       "LT".TCH_LFT_DN_REL :=         "PDI".EMO AND "PDI".EMS 
                            AND NOT "FLT".TCH_LFT_ERR 
                          //  AND     TCH_LFT_FU_RDY
                            AND NOT "PDI".LS_TCH_DN
                            AND     "PDI".LS_TEC_FLG_DN
                            AND    ("PDI".LS_TCH_SW_IN OR "PDI".LS_TCH_SW_CLN)
                            AND    "LT".TCH_SW_LOCKED
                            AND    "PDI".LS_TCH_TILT_0;

        IF "CNF_BEL_LFT_LZ550".CTRL_ACTIV = 1 THEN 

          "PDO".TCH_LFT_ENB   :=  TRUE ;  // controller enable top chamber lift


          #TCH_LFT  (Enable         := "LT".TCH_LFT_UP OR "LT".TCH_LFT_DN, 
                   CCW              := "LT".TCH_LFT_UP,   //  lift up
                   CW             := "LT".TCH_LFT_DN,   //  lift down
                   Stopp           := NOT "LT".TCH_LFT_UP AND NOT "LT".TCH_LFT_DN,
                   Reset_error     := "KYD".TCH_LFT_TRIP_RES,
                   Speed_Hz        := "CNF_TCH_LFT_LZ550".SETP,
                   PM_ADR_E        := INT_TO_WORD ("CNF_TCH_LFT_LZ550".PE_ADR),
                   PM_ADR_A        := INT_TO_WORD ("CNF_TCH_LFT_LZ550".PA_ADR)); 


        "FLT".TCH_LFT_ERR     :=  #TCH_LFT.Error;
        #TCH_LFT_FU_RDY      :=  #TCH_LFT.Ready OR "SY".SIM_ON;  
        #TCH_LFT_SPD_RCH     :=  #TCH_LFT.Speed_reached;
        #TCH_LFT_RUN         :=  #TCH_LFT.Running;    
        #TCH_LFT_ERROR_CODE  :=  #TCH_LFT.Error_code;
        #TCH_LFT_ACT_SETP    :=  #TCH_LFT.Act_Speed_Hz;

        END_IF; 

      // top chamber swivel in / out release   
      //----------------------------------------------------------------------
       "CM_ITL_IO"(ADR := 47,                                
             KYD_ON := "KYD".TCH_SW_UNLOCK AND "PDI".MP_ENB_K9,
             KYD_OFF := NOT "KYD".TCH_SW_UNLOCK OR NOT "PDI".MP_ENB_K9,
             AUTO := "APC".AUTOMATIC,
             DC_ON := "SysLog0",
             CON1 := "PDI".EMO AND "PDI".EMS,
             CON2 := "PDI".LS_GCH_UP,
             CON3 := "PDI".LS_GCH_SW_OUT,  
             CON4 := "PDI".LS_TEC_FLG_DN,   
             CON5 := "PDI".LS_TCH_TILT_0,   
             CON6 := ("PDI".LS_TCH_UP OR ("PDI".LS_TCH_DN AND ("PDI".LS_TCH_SW_CLN OR "PDI".LS_TCH_SW_OUT))),                     
             CON7 := NOT "PDO".TCH_SW_LOCK,    
             CON8 := "SysLog1",   
             ITL_OUT:= "STA_ITL_CAUSE",
             LT_OUT := "PDO".TCH_SW_UNLOCK); 

       "CM_ITL_IO"(ADR := 47,                                
             KYD_ON := ("KYD".TCH_SW_LOCK  AND "PDI".MP_ENB_K9) OR #auto_tch_sw_lock,
             KYD_OFF := (NOT "KYD".TCH_SW_LOCK OR NOT "PDI".MP_ENB_K9) AND NOT #auto_tch_sw_lock,
             AUTO := "APC".AUTOMATIC,
             DC_ON := "SysLog0",
             CON1 := "PDI".EMO AND "PDI".EMS,
             CON2 := "PDI".LS_GCH_UP,
             CON3 := "PDI".LS_GCH_SW_OUT,  
             CON4 := "PDI".LS_TEC_FLG_DN,   
             CON5 := "PDI".LS_TCH_TILT_0,   
             CON6 := ("PDI".LS_TCH_UP OR ("PDI".LS_TCH_DN AND ("PDI".LS_TCH_SW_CLN OR "PDI".LS_TCH_SW_OUT))),                     
             CON7 := NOT "PDO".TCH_SW_UNLOCK,    
             CON8 := "SysLog1",   
             ITL_OUT:= "STA_ITL_CAUSE",
             LT_OUT := "PDO".TCH_SW_LOCK); 

      IF ("PDI".LS_TCH_SW_IN OR  "PDI".LS_TCH_SW_CLN OR "PDI".LS_TCH_SW_OUT) AND NOT #fl_tch_sw_lock THEN 
         #auto_tch_sw_lock := TRUE; 
         #fl_tch_sw_lock   := TRUE;                
      ELSE
         IF #auto_tch_sw_lock AND "PDI".LS_TCH_SW_LOCK THEN
            #auto_tch_sw_lock := FALSE;
         END_IF;   
         IF NOT "PDI".LS_TCH_SW_IN AND NOT "PDI".LS_TCH_SW_CLN AND NOT "PDI".LS_TCH_SW_OUT THEN
            #fl_tch_sw_lock   :=  FALSE;
         END_IF;
      END_IF;

      "LT".TCH_SW_OUT_REL  :=  "PDI".LS_GCH_UP AND "PDI".LS_TEC_FLG_DN AND "PDI".LS_TCH_TILT_0
                             AND ("PDI".LS_TCH_UP OR ("PDI".LS_TCH_DN AND ("PDI".LS_TCH_SW_CLN OR "PDI".LS_TCH_SW_OUT))); 
      "LT".TCH_SW_IN_REL   :=  "LT".TCH_SW_OUT_REL;

      //  top chamber light signal unlock and locked 
      "LT".TCH_SW_UNLOCK      :=   NOT "PDI".LS_TCH_SW_LOCK;
      "LT".TCH_SW_LOCKED      :=   "PDI".LS_TCH_SW_LOCK;

      //----------------------------------------------------------------------
      //Top chamber tilt drive
      //----------------------------------------------------------------------
      // top chamber tilt from 0?to 30?  
       "CM_ITL_IO"(ADR := 48,                                
             KYD_ON := "KYD".TCH_TILT_30  AND "PDI".MP_ENB_K9,
             KYD_OFF := NOT "KYD".TCH_TILT_30  OR NOT "PDI".MP_ENB_K9,
             AUTO := "APC".AUTOMATIC,
             DC_ON := "SysLog0",
             CON1 := "PDI".EMO AND "PDI".EMS,
             CON2 := NOT "FLT".TCH_TILT_ERR,
             CON3 := NOT "LT".TCH_TILT_0, 
             CON4 := "PDI".LS_TCH_SW_CLN,   
             CON5 := NOT "PDI".LS_TCH_TILT_30,   
             CON6 := "PDI".LS_TCH_SW_LOCK,                     
             CON7 := "PDI".LS_TCH_UP,    
             CON8 := "SysLog1",   
             ITL_OUT := "STA_ITL_CAUSE",
             LT_OUT := "LT".TCH_TILT_30); 


       "LT".TCH_TILT_30_REL :=          "PDI".EMO AND "PDI".EMS
                              AND NOT "FLT".TCH_TILT_ERR
                            //  AND     TCH_TILT_FU_RDY 
                              AND     "PDI".LS_TCH_SW_CLN   
                              AND NOT "PDI".LS_TCH_TILT_30   
                              AND     "PDI".LS_TCH_SW_LOCK
                              AND     "PDI".LS_TCH_UP;    


       // top chamber tilt from 30?to 0?  

        "CM_ITL_IO"(ADR := 49,                                
             KYD_ON := "KYD".TCH_TILT_0 AND "PDI".MP_ENB_K9,
             KYD_OFF := NOT "KYD".TCH_TILT_0 OR NOT "PDI".MP_ENB_K9,
             AUTO := "APC".AUTOMATIC,
             DC_ON := "SysLog0",
             CON1 := "PDI".EMO AND "PDI".EMS,
             CON2 := NOT "FLT".TCH_TILT_ERR,
             CON3 := NOT "LT".TCH_TILT_30, 
             CON4 := "PDI".LS_TCH_SW_CLN,   
             CON5 := NOT "PDI".LS_TCH_TILT_0,   
             CON6 := "PDI".LS_TCH_SW_LOCK,                     
             CON7 := "SysLog1",    
             CON8 := "SysLog1",   
             ITL_OUT := "STA_ITL_CAUSE",
             LT_OUT := "LT".TCH_TILT_0); 


       "LT".TCH_TILT_0_REL :=          "PDI".EMO AND "PDI".EMS
                             AND NOT "FLT".TCH_TILT_ERR
                          //   AND     TCH_TILT_FU_RDY 
                             AND     "PDI".LS_TCH_SW_CLN   
                             AND NOT "PDI".LS_TCH_TILT_0   
                             AND     "PDI".LS_TCH_SW_LOCK;    

          IF   "CNF_TCH_TILT_LZ550".CTRL_ACTIV = 1 THEN   

               "PDO".TCH_TILT_ENB   :=  TRUE; 

      #TCH_TILT  (Enable         := "LT".TCH_TILT_0 OR "LT".TCH_TILT_30, 
                   CCW              := "LT".TCH_TILT_0,   //  tilt from 30? to 0?
                   CW               := "LT".TCH_TILT_30,   //   tilt from 0?to 30?
                   Stopp           := NOT "LT".TCH_TILT_30 AND NOT "LT".TCH_TILT_0,
                   Reset_error     := "KYD".TCH_TILT_TRIP_RES,
                   Speed_Hz        := "CNF_TCH_TILT_LZ550".SETP,
                   PM_ADR_E        := INT_TO_WORD ("CNF_TCH_TILT_LZ550".PE_ADR),
                   PM_ADR_A        := INT_TO_WORD ("CNF_TCH_TILT_LZ550".PA_ADR)); 


        "FLT".TCH_TILT_ERR     :=  #TCH_TILT.Error;
        #TCH_TILT_FU_RDY      :=  #TCH_TILT.Ready OR "SY".SIM_ON;  
        #TCH_TILT_SPD_RCH     :=  #TCH_TILT.Speed_reached;
        #TCH_TILT_RUN         :=  #TCH_TILT.Running;    
        #TCH_TILT_ERROR_CODE  :=  #TCH_TILT.Error_code;
        #TCH_TILT_ACT_SETP    :=  #TCH_TILT.Act_Speed_Hz;

        END_IF;

      //----------------------------------------------------------------------
      //technology Flange lift drive
      //----------------------------------------------------------------------
      // technology Flange lift up   

      "CM_ITL_IO"(ADR := 50,                                
             KYD_ON := "KYD".TEC_FLG_LFT_UP AND "PDI".MP_ENB_K9,
             KYD_OFF := NOT "KYD".TEC_FLG_LFT_UP OR NOT "PDI".MP_ENB_K9,
             AUTO := "APC".AUTOMATIC,
             DC_ON := "SysLog0",
             CON1 := "PDI".EMO AND "PDI".EMS,
             CON2 := NOT "FLT".TEC_FLG_LFT_ERR,
             CON3 := NOT "LT".TEC_FLG_LFT_DN, 
             CON4 := "PDI".LS_TCH_SW_OUT OR ("PDI".LS_TCH_SW_CLN AND "PDI".LS_TCH_UP),   
             CON5 := ("AV".TEC_FLG_ENC_POS < "CNF".TEC_FLG_MAX_POS),  
             CON6 := "PDI".TEC_FLG_SDL_NUT AND "PDI".SLS_TEC_FLG_LFT,                        
             CON7 := NOT #tec_flg_sw_unlock,    
             CON8 := (("AV".TEC_FLG_SW_ENC_POS<10.0) OR "DV".MP_SERVICE) AND ("PDI".LS_FCH_LFT_DN OR "DV".MP_SERVICE),   
             ITL_OUT := "STA_ITL_CAUSE",
             LT_OUT := "LT".TEC_FLG_LFT_UP); 

       "LT".TEC_FLG_LFT_UP_REL :=        "PDI".EMO AND "PDI".EMS 
                               AND NOT "FLT".TEC_FLG_LFT_ERR 
                               AND NOT "LT".TEC_FLG_LFT_DN
                               AND    ( "PDI".LS_TCH_SW_OUT OR ("PDI".LS_TCH_SW_CLN AND "PDI".LS_TCH_UP))
                               AND ("AV".TEC_FLG_ENC_POS< "CNF".TEC_FLG_MAX_POS) 
                               AND     "PDI".TEC_FLG_SDL_NUT  AND "PDI".SLS_TEC_FLG_LFT
                               AND NOT #tec_flg_sw_unlock
                               AND (("AV".TEC_FLG_SW_ENC_POS<10.0) OR "DV".MP_SERVICE) AND ("PDI".LS_FCH_LFT_DN OR "DV".MP_SERVICE); 

       // technology Flange lift down

      "CM_ITL_IO"(ADR := 51,                                
             KYD_ON := "KYD".TEC_FLG_LFT_DN AND "PDI".MP_ENB_K9,
             KYD_OFF := NOT "KYD".TEC_FLG_LFT_DN OR NOT "PDI".MP_ENB_K9,
             AUTO := "APC".AUTOMATIC,
             DC_ON := "SysLog0",
             CON1 := "PDI".EMO AND "PDI".EMS,
             CON2 := NOT "FLT".TEC_FLG_LFT_ERR,
             CON3 := NOT "LT".TEC_FLG_LFT_UP, 
             CON4 := NOT "PDI".LS_TEC_FLG_DN,   
             CON5 := "PDI".TEC_FLG_SDL_NUT AND "PDI".SLS_TEC_FLG_LFT,   
             CON6 := NOT #tec_flg_sw_unlock OR "DV".MP_SERVICE,                     
             CON7 := ("PDI".LS_FCH_LFT_DN  OR "DV".MP_SERVICE),    
             CON8 := (("AV".TEC_FLG_SW_ENC_POS<10.0) OR "DV".MP_SERVICE),   
             ITL_OUT:= "STA_ITL_CAUSE",
             LT_OUT := "LT".TEC_FLG_LFT_DN);     

       "LT".TEC_FLG_LFT_DN_REL := "PDI".EMO AND "PDI".EMS
                                AND NOT "FLT".TEC_FLG_LFT_ERR
                                AND NOT "LT".TEC_FLG_LFT_UP 
                                AND NOT "PDI".LS_TEC_FLG_DN   
                                AND "PDI".TEC_FLG_SDL_NUT AND "PDI".SLS_TEC_FLG_LFT   
                                AND (NOT #tec_flg_sw_unlock OR "DV".MP_SERVICE)                     
                                AND ("PDI".LS_FCH_LFT_DN  OR "DV".MP_SERVICE)   
                                AND (("AV".TEC_FLG_SW_ENC_POS<10.0) OR "DV".MP_SERVICE);

        IF   "CNF_TCH_TILT_LZ550".CTRL_ACTIV = 1 THEN   

               "PDO".TEC_FLG_LFT_ENB   :=  TRUE; 

        IF ("AV".TEC_FLG_ENC_POS >40.0) AND ("AV".TEC_FLG_ENC_POS < ("CNF".TEC_FLG_MAX_POS-15.0))  THEN
           IF #TEC_FLG_SET_SPD< "CNF_TEC_FLG_LFT_LZ550".SETP_FST THEN 
              #TEC_FLG_SET_SPD := #TEC_FLG_SET_SPD +1.0;
           END_IF;   
        ELSE   
           #TEC_FLG_SET_SPD := "CNF_TEC_FLG_LFT_LZ550".SETP;
        END_IF;   

        #TEC_FLG_LFT(Enable      := "LT".TEC_FLG_LFT_UP OR "LT".TEC_FLG_LFT_DN, 
                   CCW           := "LT".TEC_FLG_LFT_UP,   //  lift up
                   CW          := "LT".TEC_FLG_LFT_DN,   //  lift down
                   Stopp        := NOT "LT".TEC_FLG_LFT_UP AND NOT "LT".TEC_FLG_LFT_DN,
                   Reset_error  := "KYD".TEC_FLG_LFT_TRIP_RES,
                   Speed_Hz     := #TEC_FLG_SET_SPD,
                   PM_ADR_E     := INT_TO_WORD ("CNF_TEC_FLG_LFT_LZ550".PE_ADR),
                   PM_ADR_A     := INT_TO_WORD ("CNF_TEC_FLG_LFT_LZ550".PA_ADR)); 


        "FLT".TEC_FLG_LFT_ERR     :=  #TEC_FLG_LFT.Error;
        #TEC_FLG_LFT_FU_RDY      :=  #TEC_FLG_LFT.Ready OR "SY".SIM_ON;  
        #TEC_FLG_LFT_SPD_RCH     :=  #TEC_FLG_LFT.Speed_reached;
        #TEC_FLG_LFT_RUN         :=  #TEC_FLG_LFT.Running;    
        #TEC_FLG_LFT_ERROR_CODE  :=  #TEC_FLG_LFT.Error_code;
        #TEC_FLG_LFT_ACT_SETP    :=  #TEC_FLG_LFT.Act_Speed_Hz;

          END_IF;     

      // technology Flange swivel   
      //----------------------------------------------------------------------
      // technology Flange swivel   
      "CM_ITL_IO"(ADR := 52,                                
             KYD_ON := ("KYD".TEC_FLG_SW_UNLOCK OR #kyd_up_fch_unlock) AND "PDI".MP_ENB_K9,
             KYD_OFF := (#BI_TMR_TEC_FLG_SW> #DELAY_FCH_SW_BRK_OFF), //Close brake by 5s without movement
             AUTO := "APC".AUTOMATIC,
             DC_ON := "SysLog0",
             CON1 := "PDI".EMO AND "PDI".EMS,
             CON2 := "PDI".LS_TCH_SW_LOCK, 
             CON3 := "PDI".LS_TCH_SW_OUT,
             CON4 := NOT "PDI".LS_TEC_FLG_DN,
             CON5 := NOT "LT".TEC_FLG_LFT_UP AND NOT "LT".TEC_FLG_LFT_DN,
             CON6 := NOT "LT".FCH_LFT_UP AND NOT "LT".FCH_LFT_DN,    
             CON7 := (("AV".TEC_FLG_ENC_POS> "CNF".TEC_FLG_REL_SW_POS) OR "LT".UP_FCH_SW_UNLOCK),
             CON8 := "SysLog1",   
             ITL_OUT := "STA_ITL_CAUSE",
             LT_OUT := #tec_flg_sw_unlock);

      "PDO".TEC_FLG_SW_BRK  :=  #tec_flg_sw_unlock 
                              OR (("AV".TEC_FLG_SW_ENC_POS<5.0) AND ("AV".TEC_FLG_ENC_POS< "CNF".TEC_FLG_OP_BRK_POS) AND ("LT".TEC_FLG_LFT_DN OR "LT".FCH_LFT_DN));   

      //start opening time brake techn.flange swivel   
      //-----------------------------------------------------
      IF ABS("AV".TEC_FLG_SW_ENC_POS- "AV".UP_FCH_SW_ENC_POS)<2.0 AND ("AV".TEC_FLG_ENC_POS>30.0) AND ("AV".TEC_FLG_ENC_POS<50.0) THEN  
         #kyd_up_fch_unlock := "KYD".UP_FCH_SW_UNLOCK;
      ELSE
         #kyd_up_fch_unlock := FALSE;    
      END_IF;

      IF ABS("AV".TEC_FLG_SW_ENC_POS-#OLD_TEC_FLG_SW_POS)> 2.0 THEN   // check encoder pos. no movement
         #OLD_TEC_FLG_SW_POS  := "AV".TEC_FLG_SW_ENC_POS;
         #BI_TMR_TEC_FLG_SW   := 0;
      ELSE
         IF "PDO".TEC_FLG_SW_BRK THEN
           IF "SysTick1s" THEN 
             #BI_TMR_TEC_FLG_SW := #BI_TMR_TEC_FLG_SW + 1;
           END_IF;
         ELSE  
           #BI_TMR_TEC_FLG_SW   := 0;
         END_IF;
      END_IF;


      "LT".TEC_FLG_SW_OUT_REL  := "PDI".LS_TCH_SW_LOCK AND "PDI".LS_TCH_SW_OUT AND NOT "PDI".LS_TEC_FLG_DN AND 
                                ("AV".TEC_FLG_ENC_POS> "CNF".TEC_FLG_REL_SW_POS) AND   
                                NOT "LT".TEC_FLG_LFT_UP AND NOT "LT".TEC_FLG_LFT_DN AND NOT "LT".FCH_LFT_UP AND NOT "LT".FCH_LFT_DN ;                           
      "LT".TEC_FLG_SW_IN_REL   := "LT".TEC_FLG_SW_OUT_REL;

      //  technology flange light signal unlock
      "LT".TEC_FLG_SW_UNLOCK   := "PDO".TEC_FLG_SW_BRK;

      //----------------------------------------------------------------------
      //furnace chamber lift drive
      //----------------------------------------------------------------------
      //furnace chamber lift up   
      "CM_ITL_IO"(ADR := 53,                                
             KYD_ON := "KYD".FCH_LFT_UP AND "PDI".MP_ENB_K9,
             KYD_OFF := NOT "KYD".FCH_LFT_UP OR NOT "PDI".MP_ENB_K9,
             AUTO := "APC".AUTOMATIC,
             DC_ON := "SysLog0",
             CON1 := "PDI".EMO AND "PDI".EMS,
             CON2 := NOT "FLT".FCH_LFT_ERR,
             CON3 := NOT "LT".FCH_LFT_DN, 
             CON4 := "PDI".FCH_LFT_SDL_NUT AND "PDI".SLS_FCH_LFT,
             CON5 := ("DV".HOOK_POS_0 OR "DV".HOOK_POS_90) OR "DV".MP_SERVICE,
             CON6 := ("AV".TEC_FLG_ENC_POS> "CNF".TEC_FLG_REL_DRV_POS) AND (("AV".TEC_FLG_ENC_POS<"CNF".TEC_FLG_REL_DRV_POS+20) OR ("AV".TEC_FLG_SW_ENC_POS>50.0)),   
             CON7 := ("AV".FCH_ENC_POS< "CNF".FCH_LFT_MAX_POS),    
             CON8 := NOT #tec_flg_sw_unlock AND NOT #up_fch_sw_unlock AND NOT #lo_fch_sw_unlock,   
             ITL_OUT := "STA_ITL_CAUSE",
             LT_OUT := "LT".FCH_LFT_UP);


       "LT".FCH_LFT_UP_REL :=      "PDI".EMO AND "PDI".EMS
                             AND NOT "FLT".FCH_LFT_ERR
                             AND "PDI".FCH_LFT_SDL_NUT  AND "PDI".SLS_FCH_LFT
                             AND ("DV".HOOK_POS_0 OR "DV".HOOK_POS_90)
                             AND ("AV".TEC_FLG_ENC_POS> "CNF".TEC_FLG_REL_DRV_POS) 
                             AND (("AV".TEC_FLG_ENC_POS<"CNF".TEC_FLG_REL_DRV_POS+20) OR ("AV".TEC_FLG_SW_ENC_POS>50.0))  
                             AND ("AV".FCH_ENC_POS< "CNF".FCH_LFT_MAX_POS)
                             AND NOT #tec_flg_sw_unlock AND NOT #up_fch_sw_unlock AND NOT #lo_fch_sw_unlock;   


       // furnace chamber lift down
       "CM_ITL_IO"(ADR := 54,                                
             KYD_ON := "KYD".FCH_LFT_DN AND "PDI".MP_ENB_K9,
             KYD_OFF := NOT "KYD".FCH_LFT_DN OR NOT "PDI".MP_ENB_K9,
             AUTO := "APC".AUTOMATIC,
             DC_ON := "SysLog0",
             CON1 := "PDI".EMO AND "PDI".EMS,
             CON2 := NOT "FLT".FCH_LFT_ERR,
             CON3 := NOT "LT".FCH_LFT_UP, 
             CON4 := "PDI".FCH_LFT_SDL_NUT AND "PDI".SLS_FCH_LFT, // AND (AV.FCH_ENC_POS >= 0.0),
             CON5 := (("DV".HOOK_POS_0 OR "DV".MP_SERVICE) AND ("PDI".LS_MAG_LFT_DN OR "DV".MP_SERVICE)) OR "DV".HOOK_POS_90,
             CON6 := ("AV".TEC_FLG_ENC_POS> "CNF".TEC_FLG_REL_DRV_POS),   
             CON7 := NOT "PDI".LS_FCH_LFT_DN, 
             CON8 := NOT #tec_flg_sw_unlock AND NOT #up_fch_sw_unlock AND NOT #lo_fch_sw_unlock,   
             ITL_OUT:= "STA_ITL_CAUSE",
             LT_OUT := "LT".FCH_LFT_DN);     

       "LT".FCH_LFT_DN_REL :=     "PDI".EMO AND "PDI".EMS 
                            AND NOT "FLT".FCH_LFT_ERR
                           // AND FCH_LFT_FU_RDY
                            AND "PDI".FCH_LFT_SDL_NUT AND "PDI".SLS_FCH_LFT
                            AND (("DV".HOOK_POS_0 AND ("PDI".LS_MAG_LFT_DN OR "DV".MP_SERVICE)) OR "DV".HOOK_POS_90)
                            AND ("AV".TEC_FLG_ENC_POS> "CNF".TEC_FLG_REL_DRV_POS)
                            AND NOT "PDI".LS_FCH_LFT_DN
                            AND NOT #tec_flg_sw_unlock AND NOT #up_fch_sw_unlock AND NOT #lo_fch_sw_unlock;   

      IF "CNF_FCH_LFT_LZ550".CTRL_ACTIV = 1 THEN 

        "PDO".FCH_LFT_ENB   :=  TRUE;

        IF ("AV".FCH_ENC_POS >40.0) AND ("AV".FCH_ENC_POS < ("CNF".FCH_LFT_MAX_POS-40.0))  THEN
           IF (#FCH_LFT_SET_SPD< "CNF_FCH_LFT_LZ550".SETP_FST) AND (("AV".FCH_ENC_POS >70.0) OR "PDI".LS_FCH_HOOK_HOME) THEN 
              #FCH_LFT_SET_SPD := #FCH_LFT_SET_SPD +1.0;
           END_IF;   
        ELSE   
           #FCH_LFT_SET_SPD := "CNF_FCH_LFT_LZ550".SETP;
        END_IF;   


        #FCH_LFT(Enable         := "LT".FCH_LFT_UP OR "LT".FCH_LFT_DN, 
                   CW          := "LT".FCH_LFT_UP,   //  lift up
                   CCW         := "LT".FCH_LFT_DN,   //  lift down
                   Stopp       := NOT "LT".FCH_LFT_UP  AND NOT "LT".FCH_LFT_DN,
                   Reset_error := "KYD".FCH_LFT_TRIP_RES,
                   Speed_Hz    := #FCH_LFT_SET_SPD, // 20.0,//CNF_FCH_LFT_LZ550.SETP,
                   PM_ADR_E    := INT_TO_WORD ("CNF_FCH_LFT_LZ550".PE_ADR),
                   PM_ADR_A    := INT_TO_WORD ("CNF_FCH_LFT_LZ550".PA_ADR)); 


        "FLT".FCH_LFT_ERR     :=  #FCH_LFT.Error;
        #FCH_LFT_FU_RDY      :=  #FCH_LFT.Ready OR "SY".SIM_ON;  
        #FCH_LFT_SPD_RCH     :=  #FCH_LFT.Speed_reached;
        #FCH_LFT_RUN         :=  #FCH_LFT.Running;    
        #FCH_LFT_ERROR_CODE  :=  #FCH_LFT.Error_code;
        #FCH_LFT_ACT_SETP    :=  #FCH_LFT.Act_Speed_Hz; 

        END_IF;

      // upper furnace chamber Flange swivel   
      //----------------------------------------------------------------------
      "CM_ITL_IO"(ADR := 55,                                
             KYD_ON := "KYD".UP_FCH_SW_UNLOCK AND "PDI".MP_ENB_K9,
             KYD_OFF := (#BI_TMR_UP_FCH_SW> #DELAY_FCH_SW_BRK_OFF), //Close brake by 5s without movement
             AUTO := "APC".AUTOMATIC,
             DC_ON := "SysLog0",
             CON1 := "PDI".EMO AND "PDI".EMS,
             CON2 := ("AV".FCH_ENC_POS>"CNF".FCH_REL_SW_POS), 
             CON3 := NOT "LT".FCH_LFT_UP AND NOT "LT".FCH_LFT_DN,
             CON4 := "SysLog1",
             CON5 := "SysLog1",
             CON6 := "SysLog1",    
             CON7 := "SysLog1",
             CON8 := "SysLog1",   
             ITL_OUT := "STA_ITL_CAUSE",
             LT_OUT := #up_fch_sw_unlock);

      "PDO".UP_FCH_SW_BRK  :=  #up_fch_sw_unlock   
                             OR (("AV".UP_FCH_SW_ENC_POS<2.0) AND ("AV".FCH_ENC_POS< "CNF".UP_FCH_OP_BRK_POS) AND "LT".FCH_LFT_DN);   


      //start opening time brake upper furnace swivel   
      //-----------------------------------------------------
      IF ABS("AV".UP_FCH_SW_ENC_POS-#OLD_UP_FCH_SW_POS)> 2.0 THEN                        // check encoder pos. no movement
         #OLD_UP_FCH_SW_POS  := "AV".UP_FCH_SW_ENC_POS;
         #BI_TMR_UP_FCH_SW   := 0;
      ELSE
         IF "PDO".UP_FCH_SW_BRK THEN
           IF "SysTick1s" THEN 
             #BI_TMR_UP_FCH_SW := #BI_TMR_UP_FCH_SW + 1;
           END_IF;
         ELSE  
           #BI_TMR_UP_FCH_SW   := 0;
         END_IF;
      END_IF;

      "LT".UP_FCH_SW_OUT_REL  := ("AV".FCH_ENC_POS>"CNF".FCH_REL_SW_POS) AND NOT "LT".FCH_LFT_UP AND NOT "LT".FCH_LFT_DN;                            
      "LT".UP_FCH_SW_IN_REL   := "LT".UP_FCH_SW_OUT_REL;

      // upper furnace chamber light signal unlock
      "LT".UP_FCH_SW_UNLOCK   := "PDO".UP_FCH_SW_BRK;


      // lower furnace chamber Flange swivel   
      //----------------------------------------------------------------------
      "CM_ITL_IO"(ADR := 56,                                
             KYD_ON := "KYD".LO_FCH_SW_UNLOCK AND "PDI".MP_ENB_K9,
             KYD_OFF := (#BI_TMR_LO_FCH_SW> #DELAY_FCH_SW_BRK_OFF), //Close brake by 3s without movement
             AUTO := "APC".AUTOMATIC,
             DC_ON := "SysLog0",
             CON1 := "PDI".EMO AND "PDI".EMS,
             CON2 := ("PDI".LS_FCH_LFT_DN OR (("AV".FCH_ENC_POS>"CNF".FCH_REL_SW_POS) AND "LT".FCH_HOOK_WORK)), 
             CON3 := "PDI".LS_MAG_LFT_DN OR "DV".MP_SERVICE,
             CON4 := NOT "LT".FCH_LFT_UP AND NOT "LT".FCH_LFT_DN,
             CON5 := "SysLog1",
             CON6 := "SysLog1",    
             CON7 := "SysLog1",
             CON8 := "SysLog1",   
             ITL_OUT := "STA_ITL_CAUSE",
             LT_OUT := #lo_fch_sw_unlock);

      "PDO".LO_FCH_SW_BRK  :=  #lo_fch_sw_unlock   
                             OR (("AV".LO_FCH_SW_ENC_POS<2.0) AND ("AV".FCH_ENC_POS< "CNF".LO_FCH_OP_BRK_POS) AND "LT".FCH_LFT_DN);   

      //start opening time brake lower furnace swivel   
      //-----------------------------------------------------
      IF ABS("AV".LO_FCH_SW_ENC_POS-#OLD_LO_FCH_SW_POS)> 2.0 THEN                        // check encoder pos. no movement
         #OLD_LO_FCH_SW_POS  := "AV".LO_FCH_SW_ENC_POS;
         #BI_TMR_LO_FCH_SW   := 0;
      ELSE
         IF "PDO".LO_FCH_SW_BRK THEN
           IF "SysTick1s" THEN 
             #BI_TMR_LO_FCH_SW := #BI_TMR_LO_FCH_SW + 1;
           END_IF;
         ELSE  
           #BI_TMR_LO_FCH_SW   := 0;
         END_IF;
      END_IF;

       "LT".LO_FCH_SW_OUT_REL  :=  ("PDI".LS_FCH_LFT_DN OR (("AV".FCH_ENC_POS>"CNF".FCH_REL_SW_POS) AND "LT".FCH_HOOK_WORK))AND 
                                 ("PDI".LS_MAG_LFT_DN OR "DV".MP_SERVICE) AND NOT "LT".FCH_LFT_UP AND NOT "LT".FCH_LFT_DN ;  
       "LT".LO_FCH_SW_IN_REL   :=  "LT".LO_FCH_SW_OUT_REL;

      // lower furnace chamber light signal unlock
      "LT".LO_FCH_SW_UNLOCK   := "PDO".LO_FCH_SW_BRK;


      //----------------------------------------------------------------------
      //furnace chamber hook
      //----------------------------------------------------------------------
      // furnace chamber hook home pos 

      "CM_ITL_IO"(ADR := 57,                                
             KYD_ON := "KYD".FCH_HOOK_HOME AND "PDI".MP_ENB_K9,
             KYD_OFF := NOT "KYD".FCH_HOOK_HOME OR NOT "PDI".MP_ENB_K9,
             AUTO := "APC".AUTOMATIC,
             DC_ON := "SysLog0",
             CON1 := "PDI".EMO AND "PDI".EMS,
             CON2 := "PDI".LS_MAG_LFT_DN,
             CON3 := "PDI".LS_FCH_LFT_DN,
             CON4 := "DV".HOOK_POS_0,
             CON5 := NOT "PDO".LO_FCH_SW_BRK,     
             CON6 := NOT "PDI".LS_FCH_HOOK_HOME,                     
             CON7 := "SysLog1",    
             CON8 := "SysLog1", 
             ITL_OUT := "STA_ITL_CAUSE",
             LT_OUT := "PDO".FCH_HOOK_HOME);

      "LT".FCH_HOOK_HOME := "PDI".LS_FCH_HOOK_HOME; //PDO.FCH_HOOK_HOME;

      "LT".FCH_HOOK_HOME_REL  :=      "PDI".EMO AND "PDI".EMS
                                AND "PDI".LS_MAG_LFT_DN
                                AND "PDI".LS_FCH_LFT_DN
                                AND "DV".HOOK_POS_0
                                AND NOT "PDO".LO_FCH_SW_BRK
                                AND NOT "PDI".LS_FCH_HOOK_HOME;


      // furnace chamber hook working pos 

      "CM_ITL_IO"(ADR := 58,                                
             KYD_ON := "KYD".FCH_HOOK_WORK AND "PDI".MP_ENB_K9,
             KYD_OFF := NOT "KYD".FCH_HOOK_WORK OR NOT "PDI".MP_ENB_K9,
             AUTO := "APC".AUTOMATIC,
             DC_ON := "SysLog0",
             CON1 := "PDI".EMO AND "PDI".EMS,
             CON2 := "PDI".LS_MAG_LFT_DN,
             CON3 := "PDI".LS_FCH_LFT_DN,
             CON4 := "DV".HOOK_POS_0,
             CON5 := NOT "PDO".LO_FCH_SW_BRK,     
             CON6 := NOT "PDI".LS_FCH_HOOK_WORK,                     
             CON7 := "SysLog1",    
             CON8 := "SysLog1", 
             ITL_OUT := "STA_ITL_CAUSE",
             LT_OUT := "PDO".FCH_HOOK_WORK);

       "LT".FCH_HOOK_WORK := "PDI".LS_FCH_HOOK_WORK; //PDO.FCH_HOOK_WORK;


       "LT".FCH_HOOK_WORK_REL  :=     "PDI".EMO AND "PDI".EMS
                                AND "PDI".LS_MAG_LFT_DN
                                AND "PDI".LS_FCH_LFT_DN
                                AND "DV".HOOK_POS_0
                                AND NOT "PDO".LO_FCH_SW_BRK
                                AND NOT "PDI".LS_FCH_HOOK_WORK;

       //----------------------------------------------------------------------
       //  magnet lift drive
       //----------------------------------------------------------------------
           // Magnet downwards
          "CM_ITL_IO"(ADR := 59,
                 KYD_ON := "KYD".MAG_DRV_DN AND ("PDI".MP_ENB_K5 OR "PDI".MP_ENB_K9),
                 KYD_OFF:= NOT "KYD".MAG_DRV_DN OR (NOT "PDI".MP_ENB_K5 AND NOT "PDI".MP_ENB_K9),
                 AUTO := "APC".AUTOMATIC,
                 DC_ON:= "SysLog0",
                 CON1 := "PDI".EMO AND "PDI".EMS,
                 CON2 := NOT "LT".MAG_ON,
                 CON3 := NOT "PDI".LS_MAG_LFT_DN,                         
                 CON4 := NOT "FLT".MAG_LFT_SDL_ERR,    
                 CON5 := "PDI".SLS_MAG_LFT,               
                 CON6 := "DV".HOOK_POS_90 OR "DV".MP_SERVICE,
                 CON7 := NOT "PDO".LO_FCH_SW_BRK,                       
                 CON8 := "SysLog1",
                 ITL_OUT:= "STA_ITL_CAUSE",
                 LT_OUT := "LT".MAG_LFT_DN);

        "LT".MAG_LFT_DN_REL  :=        "PDI".EMO AND "PDI".EMS
                             AND NOT "LT".MAG_ON
                             AND NOT "PDI".LS_MAG_LFT_DN
                             AND NOT "FLT".MAG_LFT_SDL_ERR                        
                             AND     "PDI".SLS_MAG_LFT   
                             AND     ("DV".HOOK_POS_90 OR "DV".MP_SERVICE)
                             AND NOT "PDO".LO_FCH_SW_BRK;

       // Magnet upwards
          "CM_ITL_IO"(ADR := 60,
                 KYD_ON := "KYD".MAG_DRV_UP AND ("PDI".MP_ENB_K5 OR "PDI".MP_ENB_K9),
                 KYD_OFF:= NOT "KYD".MAG_DRV_UP OR (NOT "PDI".MP_ENB_K5 AND NOT "PDI".MP_ENB_K9),
                 AUTO := "APC".AUTOMATIC,
                 DC_ON:= "SysLog0",
                 CON1 := "PDI".EMO AND "PDI".EMS,
                 CON2 := NOT "LT".MAG_ON,
                 CON3 := NOT "PDI".LS_MAG_LFT_UP,                         
                 CON4 := NOT "FLT".MAG_LFT_SDL_ERR,    
                 CON5 := "PDI".SLS_MAG_LFT,               
                 CON6 := "DV".HOOK_POS_90 OR "DV".MP_SERVICE,
                 CON7 := NOT "PDO".LO_FCH_SW_BRK,                                              
                 CON8 := "SysLog1",
                 ITL_OUT:= "STA_ITL_CAUSE",
                 LT_OUT := "LT".MAG_LFT_UP);

       "LT".MAG_LFT_UP_REL :=         "PDI".EMO AND "PDI".EMS
                             AND NOT "LT".MAG_ON
                             AND NOT "PDI".LS_MAG_LFT_UP
                             AND NOT "FLT".MAG_LFT_SDL_ERR                        
                             AND     "PDI".SLS_MAG_LFT   
                             AND     ("DV".HOOK_POS_90 OR "DV".MP_SERVICE)
                             AND NOT "PDO".LO_FCH_SW_BRK;


       "PDO".BRK_MAG_LFT := "LT".MAG_LFT_UP OR "LT".MAG_LFT_DN;
       "PDO".MAG_LFT_DN  := "LT".MAG_LFT_DN AND NOT "LT".MAG_LFT_UP;  //AND mag_drv_dly_over
       "PDO".MAG_LFT_UP  := "LT".MAG_LFT_UP AND NOT "LT".MAG_LFT_DN;  //AND mag_drv_dly_over

       //delay start of magnet lift movement
       //-----------------------------------
       #iTime := S_ODT( T_NO:= "BM_TMR_MAG_DRV",                  // Timer
                       S   := "PDO".BRK_MAG_LFT,               // Start Condition
                       TV  := #DELAY_MAG_DRV_ON,                // Time Setpoint
                       R   := NOT "PDO".BRK_MAG_LFT,           // Reset Condition
                       BI  => #BI_TMR_MAG_DRV,                  // Current Time Value
                       Q   => #mag_drv_dly_over);               // Output  


       //set warning light outputs
       //-------------------------
       "PDO".HOR_MAG_ACTIVE :=  ("PDO".MAG_LFT_DN OR "PDO".MAG_LFT_UP) AND "SysCycle2s";
       "PDO".LMP_MAG_ACTIVE :=  ("PDO".MAG_LFT_DN OR "PDO".MAG_LFT_UP) AND "SysCycle2s"; 

       //set alarms
       //----------
       "FLT".MAG_SLS := NOT "PDI".SLS_MAG_LFT; 
       "FLT".MAG_LFT_SDL_ERR :=  NOT("PDI".MAG_LFT_SDL_NUT1 AND "PDI".MAG_LFT_SDL_NUT2 AND "PDI".MAG_LFT_SDL_NUT3); 


      //-----------------------------------------------------------------------------
    //  signals for all positions of parts 

       "LT".GCH_BEL_UP   := NOT "PDI".LS_GCH_BEL_UP  AND "PDI".LS_GCH_BEL_DN;
       "LT".GCH_BEL_DN   := NOT "PDI".LS_GCH_BEL_DN  AND "PDI".LS_GCH_BEL_UP;
       IF "LT".GCH_BEL_UP THEN
          "STA".BEL_LFT_POS     := 100;
       ELSIF "LT".GCH_BEL_DN THEN
          "STA".BEL_LFT_POS     := 0;
       ELSIF "LT".BEL_LFT_UP THEN
           IF "SysTick1s" AND ("STA".BEL_LFT_POS<90) THEN
               "STA".BEL_LFT_POS := "STA".BEL_LFT_POS +5;
           END_IF;
       ELSIF "LT".BEL_LFT_DN THEN
           IF "SysTick1s" AND ("STA".BEL_LFT_POS>10) THEN
               "STA".BEL_LFT_POS := "STA".BEL_LFT_POS -5;
           END_IF;
       END_IF;


       "LT".GCH_UP       := "PDI".LS_GCH_UP      AND NOT "PDI".LS_GCH_DN;
       "LT".GCH_DN       := "PDI".LS_GCH_DN      AND NOT "PDI".LS_GCH_UP;
       IF "LT".GCH_UP THEN
          "STA".GCH_LFT_POS := 100;
       ELSIF "LT".GCH_DN THEN
          "STA".GCH_LFT_POS  := 0;
       ELSIF "LT".GCH_LFT_UP THEN
           IF "SysTick1s" AND ("STA".GCH_LFT_POS<90) THEN
               "STA".GCH_LFT_POS := "STA".GCH_LFT_POS +5;
           END_IF;
       ELSIF "LT".GCH_LFT_DN THEN
           IF "SysTick1s" AND ("STA".GCH_LFT_POS>10) THEN
               "STA".GCH_LFT_POS := "STA".GCH_LFT_POS -5;
           END_IF;
       END_IF;

       "LT".GCH_IN       := "PDI".LS_GCH_SW_IN   AND NOT "PDI".LS_GCH_SW_CLN    AND NOT "PDI".LS_GCH_SW_OUT;
       "LT".GCH_CLN      := "PDI".LS_GCH_SW_CLN  AND NOT "PDI".LS_GCH_SW_IN     AND NOT "PDI".LS_GCH_SW_OUT;
       "LT".GCH_OUT      := "PDI".LS_GCH_SW_OUT  AND NOT "PDI".LS_GCH_SW_IN     AND NOT "PDI".LS_GCH_SW_CLN;
       IF "LT".GCH_IN THEN
          "STA".GCH_SW_POS := 0;
       ELSIF "LT".GCH_CLN THEN
          "STA".GCH_SW_POS  := 50;
       ELSIF "LT".GCH_OUT THEN
          "STA".GCH_SW_POS := 100;
       ELSE
          "STA".GCH_SW_POS := 40;
       END_IF;

       "LT".TCH_UP           := "PDI".LS_TCH_UP      AND NOT "PDI".LS_TCH_DN; 
       "LT".TCH_DN           := "PDI".LS_TCH_DN      AND NOT "PDI".LS_TCH_UP; 
       IF "LT".TCH_UP THEN
          "STA".TCH_LFT_POS := 100;
       ELSIF "LT".TCH_DN THEN
          "STA".TCH_LFT_POS  := 0;
       ELSIF "LT".TCH_LFT_UP THEN
           IF "SysTick1s" AND ("STA".TCH_LFT_POS<80) THEN
               "STA".TCH_LFT_POS := "STA".TCH_LFT_POS +10;
           END_IF;
       ELSIF "LT".TCH_LFT_DN THEN
           IF "SysTick1s" AND ("STA".TCH_LFT_POS>20) THEN
               "STA".TCH_LFT_POS := "STA".TCH_LFT_POS -10;
           END_IF;
       END_IF;

       "LT".TCH_IN           := "PDI".LS_TCH_SW_IN   AND NOT "PDI".LS_TCH_SW_CLN AND NOT "PDI".LS_TCH_SW_OUT;
       "LT".TCH_CLN          := "PDI".LS_TCH_SW_CLN  AND NOT "PDI".LS_TCH_SW_IN  AND NOT "PDI".LS_TCH_SW_OUT;
       "LT".TCH_OUT          := "PDI".LS_TCH_SW_OUT  AND NOT "PDI".LS_TCH_SW_IN  AND NOT "PDI".LS_TCH_SW_CLN;
       IF "LT".TCH_IN THEN
          "STA".TCH_SW_POS := 0;
       ELSIF "LT".TCH_CLN THEN
          "STA".TCH_SW_POS  := 50;
       ELSIF "LT".TCH_OUT THEN
          "STA".TCH_SW_POS := 100;
       ELSE
          "STA".TCH_SW_POS := 40;
       END_IF;

       "LT".TCH_TILT_POS_0   := "PDI".LS_TCH_TILT_0  AND NOT "PDI".LS_TCH_TILT_30; 
       "LT".TCH_TILT_POS_30  := "PDI".LS_TCH_TILT_30 AND NOT "PDI".LS_TCH_TILT_0; 
       IF "LT".TCH_TILT_POS_0 THEN
          "STA".TCH_TILT_POS := 0;
       ELSIF "LT".TCH_TILT_POS_30 THEN
          "STA".TCH_TILT_POS  := 100;
       ELSE 
          "STA".TCH_TILT_POS := 15;
       END_IF;

       "LT".MAG_UP           := "PDI".LS_MAG_LFT_UP      AND NOT "PDI".LS_MAG_LFT_DN; 
       "LT".MAG_DN           := "PDI".LS_MAG_LFT_DN      AND NOT "PDI".LS_MAG_LFT_UP;
       "STA".MAG_LFT_POS     := REAL_TO_INT(100.0 * #mag_pos_cal/850.0);
       IF "PDI".LS_MAG_LFT_UP THEN
          "STA".MAG_LFT_POS := 100;
          #mag_pos_cal     := 850.0;
       ELSE 
          IF "PDI".LS_MAG_LFT_DN THEN
             "STA".MAG_LFT_POS  := 0;
             #mag_pos_cal      := 0.0;
          ELSE
             IF "LT".MAG_LFT_UP THEN
                IF "SysTick100ms" AND (#mag_pos_cal<844.5) THEN
                  #mag_pos_cal := #mag_pos_cal +0.5;
                END_IF;
             ELSE  
                IF "LT".MAG_LFT_DN THEN
                  IF "SysTick100ms" AND (#mag_pos_cal>5.5) THEN
                     #mag_pos_cal := #mag_pos_cal -0.5;                  
                  END_IF;
                ELSE
                  IF #mag_pos_cal=0 THEN
                     #mag_pos_cal := 10.0; 
                  END_IF;                        
                END_IF;
             END_IF;             
          END_IF;
       END_IF;

       //  mobil panel display actual value of position via encoder

       "DIS".ACT_TEC_FCH_SW_POS  :=  "AV".TEC_FLG_SW_ENC_POS; 
       "DIS".ACT_UP_FCH_SW_POS   :=  "AV".UP_FCH_SW_ENC_POS ; 
       "DIS".ACT_LO_FCH_SW_POS   :=  "AV".LO_FCH_SW_ENC_POS ; 

       "DIS".ACT_TEC_FLG_LFT_POS  :=  "AV".TEC_FLG_ENC_POS; 
       IF "DIS".ACT_TEC_FLG_LFT_POS< 1000.0 THEN
           "STA".TEC_FLG_POS := REAL_TO_INT("DIS".ACT_TEC_FLG_LFT_POS/10.0)+ "STA".UP_FCH_LFT_POS;        
       END_IF;    
       "DIS".ACT_FCH_LFT_POS      :=  "AV".FCH_ENC_POS; 
       IF "DIS".ACT_FCH_LFT_POS< 1000.0 THEN
           "STA".UP_FCH_LFT_POS := REAL_TO_INT("DIS".ACT_FCH_LFT_POS/10.0);
           IF "DV".HOOK_POS_0 AND "PDI".LS_FCH_HOOK_WORK THEN
               IF "STA".UP_FCH_LFT_POS>10 THEN
                  "STA".LO_FCH_LFT_POS :=  "STA".UP_FCH_LFT_POS-10;
               END_IF;
           ELSE
               "STA".LO_FCH_LFT_POS := 0; 
           END_IF;          
       END_IF;    

       // Technology flange is in home position 
       "DV".TEC_FLG_SW_HOME_POS := ABS("AV".TEC_FLG_SW_ENC_POS- "CNF".TEC_FLG_SW_HOME_POS) <2.0; 

       // upper furnace chamber is in home position 
       "DV".UP_FCH_SW_HOME_POS := ABS("AV".UP_FCH_SW_ENC_POS- "CNF".UP_FCH_SW_HOME_POS)<2.0;;

       // lower furnace chamber is in home position 
       "DV".LO_FCH_SW_HOME_POS := ABS("AV".LO_FCH_SW_ENC_POS- "CNF".LO_FCH_SW_HOME_POS)< 2.0;

       //  working position / HOOK parking
       "DV".HOOK_POS_0  :=  ABS("AV".LO_FCH_SW_ENC_POS-"CNF".LO_FCH_SW_HOME_POS)< 2.0;   // Release position -2..2?
       "DV".HOOK_POS_90 :=  ABS("AV".LO_FCH_SW_ENC_POS-"CNF".LO_FCH_SW_PARK_POS)< 2.0;   // Release position -88..92?



       //----------------------------------------------------------------------
       // V7  gate valve lift drive 
       //----------------------------------------------------------------------
       #diff_prs_ok:= (ABS("DIS".ACT_PRS_CLF-"DIS".ACT_PRS_CGT)<40.0) 
                      OR ("DV".APS_GCH_DELAYED AND "DV".APS_FCH_DELAYED);

       //V7 LIFT UP (open)
       "CM_ITL_IO"(ADR := 16,
              KYD_ON := "KYD".V7_LFT_UP AND "PDI".MP_ENB_K9,
              KYD_OFF := NOT "KYD".V7_LFT_UP OR NOT "PDI".MP_ENB_K9,
              AUTO := "APC".AUTOMATIC,
              DC_ON:= "SysLog0", 
              CON1 := "PDI".EMO AND "PDI".EMS,
              CON2 := "DV".MAIN_SWITCH_ON,
              CON3 := #diff_prs_ok,
              CON4 := NOT "PDI".LS_V7_UP,               
              CON5 := NOT "PDI".LS_V7_SW_OUT AND NOT "PDI".LS_V7_CLN_POS,//DV.LS_V7_SW_IN_DLY AND NOT PDI.LS_V7_SW_OUT AND NOT PDI.LS_V7_CLN_POS,
              CON6 := "PDI".LS_V7_SW_IN,                             
              CON7 := NOT "LT".V7_LFT_DN,                             
              CON8 := NOT "LT".V7_SW_IN AND NOT "LT".V7_SW_OUT,
              ITL_OUT:= "STA_ITL_CAUSE",
              LT_OUT := "LT".V7_LFT_UP);

       // light signal release V7 lift up    
       "LT".V7_LFT_UP_REL :=     "PDI".EMO AND "PDI".EMS 
                           AND "DV".MAIN_SWITCH_ON 
                       //    AND diff_prs_ok
                           AND NOT "PDI".LS_V7_SW_OUT 
                           AND NOT "PDI".LS_V7_UP 
                           AND NOT "PDI".LS_V7_CLN_POS
                           AND "DV".LS_V7_SW_IN_DLY 
                           AND NOT "LT".V7_SW_IN AND NOT "LT".V7_SW_OUT;     

       //V7 lift down (close)
       #rel_drv_xt_pos := "DIS".ACT_XT_POS< 3000.0;

       "CM_ITL_IO"(ADR := 17,
              KYD_ON := "KYD".V7_LFT_DN AND "PDI".MP_ENB_K9,
              KYD_OFF := NOT "KYD".V7_LFT_DN OR NOT "PDI".MP_ENB_K9,
              AUTO := "APC".AUTOMATIC,
              DC_ON:= "SysLog0",  
              CON1 := "PDI".EMO AND "PDI".EMS,
              CON2 := "DV".MAIN_SWITCH_ON,
              CON3 := NOT "PDI".LS_V7_DN,               
              CON4 := NOT "PDI".LS_V7_SW_OUT AND NOT "PDI".LS_V7_CLN_POS, //DV.LS_V7_SW_IN_DLY AND NOT PDI.LS_V7_SW_OUT AND NOT PDI.LS_V7_CLN_POS,
              CON5 := NOT "LT".V7_SW_IN,                             
              CON6 := NOT "LT".V7_LFT_UP,
              CON7 := NOT "LT".V7_SW_OUT,           
              CON8 := "DV".LS_V7_SW_IN_DLY,
              ITL_OUT:= "STA_ITL_CAUSE",
              LT_OUT := "LT".V7_LFT_DN);

       // light signal release V7 lift dn
       "LT".V7_LFT_DN_REL :=     "PDI".EMO AND "PDI".EMS
                           AND "DV".MAIN_SWITCH_ON
                           AND NOT "PDI".LS_V7_SW_OUT
                           AND NOT  "PDI".LS_V7_DN 
                           AND NOT  "PDI".LS_V7_CLN_POS              
                           AND "DV".LS_V7_SW_IN_DLY
                           AND NOT "LT".V7_SW_IN AND NOT "LT".V7_SW_OUT;      

        IF "CNF_V7_LFT_LZ550".CTRL_ACTIV = 1 THEN 

           "PDO".GTE_V_LFT_ENB   :=  TRUE;  // controller enable v7low lift



         #V7_LFT(Enable         := "LT".V7_LFT_UP OR "LT".V7_LFT_DN, 
                   CW              := "LT".V7_LFT_UP, // LT.V7_LFT_UP,   //  lift up
                   CCW             := "LT".V7_LFT_DN,   //  lift down
                   Stopp           := NOT "LT".V7_LFT_UP AND NOT "LT".V7_LFT_DN,
                   Reset_error     := "KYD".V7_LFT_TRIP_RES,
                   Speed_Hz        :=  10.0 ,     //CNF_V7_LFT_LZ550.SETP,
                   PM_ADR_E        := INT_TO_WORD ("CNF_V7_LFT_LZ550".PE_ADR),
                   PM_ADR_A        := INT_TO_WORD ("CNF_V7_LFT_LZ550".PA_ADR)); 


        "FLT".V7_LFT_ERR     :=  #V7_LFT.Error;
       // V7_LFT_FU_RDY      :=  V7_LFT.READY OR SY.SIM_ON;  
        #V7_LFT_SPD_RCH     :=  #V7_LFT.Speed_reached;
      //  V7_LFT_RUN         :=  V7_LFT.RUNNING;    
        #V7_LFT_ERROR_CODE      :=  #V7_LFT.Error_code;
        #V7_LFT_ACT_SETP        :=  #V7_LFT.Act_Speed_Hz;

       END_IF;







       //V7 swivel out 
       "CM_ITL_IO"(ADR := 18,
              KYD_ON := "KYD".V7_SW_OUT AND "PDI".MP_ENB_K9,
              KYD_OFF:= NOT "KYD".V7_SW_OUT OR NOT "PDI".MP_ENB_K9,
              AUTO := "APC".AUTOMATIC,
              DC_ON:= "SysLog0",
              CON1 := "PDI".EMO AND "PDI".EMS,
              CON2 := "DV".MAIN_SWITCH_ON,
              CON3 := "DV".LS_V7_UP_DLY,
              CON4 := (NOT "PDI".LS_V7_SW_OUT AND NOT "PDI".LS_V7_FLP_OP) OR ("PDI".LS_V7_FLP_OP AND NOT "PDI".LS_V7_CLN_POS),               
              CON5 := NOT "LT".V7_SW_IN,
              CON6 := NOT "LT".V7_LFT_UP AND NOT "LT".V7_LFT_DN,                             
              CON7 := "PDI".LS_V7_UP,                             
              CON8 := "SysLog1",
              ITL_OUT:= "STA_ITL_CAUSE",
              LT_OUT := "LT".V7_SW_OUT);

       // light signal release V7 swivel out
       "LT".V7_SW_OUT_REL :=          "PDI".EMO AND "PDI".EMS
                           AND      "DV".MAIN_SWITCH_ON
                           AND      "DV".LS_V7_UP_DLY
                           AND (NOT "PDI".LS_V7_SW_OUT AND NOT "PDI".LS_V7_FLP_OP) OR ("PDI".LS_V7_FLP_OP AND NOT "PDI".LS_V7_CLN_POS) 
                           AND NOT "LT".V7_SW_IN
                           AND NOT "LT".V7_LFT_UP 
                           AND NOT "LT".V7_LFT_DN
                           AND "PDI".LS_V7_UP;

       //V7 swivel in 
       "CM_ITL_IO"(ADR := 19,
              KYD_ON := "KYD".V7_SW_IN AND "PDI".MP_ENB_K9,
              KYD_OFF:= NOT "KYD".V7_SW_IN OR NOT "PDI".MP_ENB_K9,
              AUTO := "APC".AUTOMATIC,
              DC_ON:= "SysLog0",
              CON1 := "PDI".EMO AND "PDI".EMS,
              CON2 := "DV".MAIN_SWITCH_ON,
              CON3 := NOT "LT".V7_LFT_DN,           //DV.LS_V7_UP_DLY,
              CON4 := NOT "PDI".LS_V7_SW_IN,               
              CON5 := NOT "LT".V7_SW_OUT,
              CON6 := NOT "LT".V7_LFT_UP,                                                        
              CON7 := #rel_drv_xt_pos,    
              CON8 := "SysLog1",
              ITL_OUT:= "STA_ITL_CAUSE",
              LT_OUT := "LT".V7_SW_IN); 

       // light signal release V7 swivel in 
       "LT".V7_SW_IN_REL :=           "PDI".EMO AND "PDI".EMS
                           AND      "DV".MAIN_SWITCH_ON
                           AND NOT  "PDI".LS_V7_SW_IN               
                           AND NOT "LT".V7_LFT_UP 
                           AND NOT "LT".V7_LFT_DN
                           AND NOT "LT".V7_SW_OUT;   

        IF "CNF_V7_SW_LZ550".CTRL_ACTIV = 1 THEN 

           "PDO".GTE_V_SW_ENB   :=  TRUE;  // controller enable v7low lift



         #V7_SW(Enable         := "LT".V7_SW_IN OR "LT".V7_SW_OUT, 
                   CW              := "LT".V7_SW_IN, // LT.V7_SW_UP,   //  lift up
                   CCW             := "LT".V7_SW_OUT,   //  lift down
                   Stopp           := NOT "LT".V7_SW_IN AND NOT "LT".V7_SW_OUT,
                   Reset_error     := "KYD".V7_SW_TRIP_RES,
                   Speed_Hz        := "CNF_V7_SW_LZ550".SETP,
                   PM_ADR_E        := INT_TO_WORD ("CNF_V7_SW_LZ550".PE_ADR),
                   PM_ADR_A        := INT_TO_WORD ("CNF_V7_SW_LZ550".PA_ADR)); 


        "FLT".V7_SW_ERR     :=  #V7_SW.Error;
       // V7_SW_FU_RDY      :=  V7_SW.READY OR SY.SIM_ON;  
        #V7_SW_SPD_RCH     :=  #V7_SW.Speed_reached;
      //  V7_SW_RUN         :=  V7_SW.RUNNING;    
        #V7_SW_ERROR_CODE      :=  #V7_SW.Error_code;
        #V7_SW_ACT_SETP        :=  #V7_SW.Act_Speed_Hz;

       END_IF;


       // signal of positions
       "LT".V7_OPEN    := "PDI".LS_V7_UP AND NOT "PDI".LS_V7_DN AND "PDI".LS_V7_SW_OUT;
       "LT".V7_CLOSE   := "PDI".LS_V7_DN AND NOT "PDI".LS_V7_UP;
       "LT".V7_CLN     := "PDI".LS_V7_CLN_POS  AND NOT "PDI".LS_V7_SW_IN  AND NOT "PDI".LS_V7_SW_OUT;

       IF "LT".V7_CLOSE THEN
          "STA".V7_LFT_POS := 0;
       ELSIF NOT "PDI".LS_V7_DN AND NOT "PDI".LS_V7_UP THEN
              "STA".V7_LFT_POS := 50;
       ELSIF "PDI".LS_V7_UP THEN
          "STA".V7_LFT_POS := 100;
       END_IF;

       IF "PDI".LS_V7_SW_IN THEN
          "STA".V7_SW_POS := 0;
       ELSIF NOT "PDI".LS_V7_SW_IN AND NOT "PDI".LS_V7_SW_OUT THEN
          "STA".V7_SW_POS := 25;
       ELSIF "PDI".LS_V7_SW_OUT THEN
             "STA".V7_SW_POS := 50;           
       ELSIF "PDI".LS_V7_CLN_POS THEN
          "STA".V7_SW_POS := 100;
       END_IF;

      //------------------------------------------
      //  controller enable  
      //------------------------------------------ 

      // controller enable gate chamber lift

      // controller enable TOP chamber lift


      // controller enable TOP chamber tilt


      // controller enable technology flange lift


      // controller enable furnace chamber lift
END_FUNCTION_BLOCK

FUNCTION_BLOCK "BM_VSL_HDL_DRV"   // FB63, SCL
{ S7_Optimized_Access := 'FALSE' }
VERSION : 0.0
// --------------------------------------------------------------------------------
//     program     :   BM_VSL_HDL_DRV
//     description :   handling drives of vessel parts
//     name        :   John Wang
//     date        :   22.10.2018
//   
//     revision    :
//     name        :
//     date        :    
//                     (c)PVA CGS GmbH
//     --------------------------------------------------------------------------------
BEGIN









    ;
END_FUNCTION_BLOCK

FUNCTION_BLOCK "BM_CALL_DRV"   // FB66, SCL
{ S7_Optimized_Access := 'FALSE' }
VERSION : 0.0
// --------------------------------------------------------------------------------
//     program     :    BM_CALL_DRV
//     description :    call all drive modules 
//     name        :    K. Kalkowski
//     date        :    19.11.99
// 
//     revision    :    converter with LZi950 
//     name        :    John Wang
//     date        :    07.12.2018
//                    
//                     (c)PVA CGS GMBH
//     --------------------------------------------------------------------------------
   VAR
      BM_DRV_XT_LFT : "PM_DRV_COMM_LZI950";
      BM_DRV_XT_ROT : "PM_DRV_COMM_LZI950";
      BM_DRV_CR_LFT : "PM_DRV_COMM_LZI950";
      BM_DRV_CR_ROT : "PM_DRV_COMM_LZI950";
      set_speed_lft : Real;
      set_spd_xt_lft_real : Real;
      set_spd_xt_lft : Real;
      set_speed_rot : Real;
      set_spd_xt_rot_real : Real;
      set_spd_xt_rot : Real;
      set_speed_cr_lft : Real;
      set_spd_cr_lft_real : Real;
      set_spd_cr_lft : Real;
      set_speed_cr_rot : Real;
      xt_lft_up : Bool;
      xt_lft_dn : Bool;
      xt_rot_cw : Bool;
      xt_rot_ccw : Bool;
      cr_lft_up : Bool;
      cr_lft_dn : Bool;
      cr_rot_cw : Bool;
      cr_rot_ccw : Bool;
      Dummy : Bool;
   END_VAR
   VAR_TEMP
      out_dummy_bool : Bool;
      on_dummy : Bool;
      off_dummy : Bool;
      real_0_dummy : Real;
      int_0_dummy : Int;
      kyd_cr_lft_up : Bool;
      kyd_cr_lft_dn : Bool;
      kyd_cr_lft_fast : Bool;
      kyd_cr_lft_stop : Bool;
      cr_lft_down_enb : Bool;
      kyd_xt_lft_up : Bool;
      kyd_xt_lft_dn : Bool;
      kyd_xt_lft_fast : Bool;
      kyd_xt_lft_stop : Bool;
      xt_lft_fast : Bool;
      xt_lft_down_enb : Bool;
      cruc_rot_ctl : Bool;
      cr_rot_osci_req : Bool;
      xt_rot : Real;
      cr_rot_set : Real;
      cr_rot_act : Real;
      cr_rot_inc : Real;
      set_cr_rot_ofs : Real;
      ac_in : Real;
      gear_cr_rot : Real;
      kya_cruc_rot_set_in : Real;
      kya_set_xt_lft : Real;
      kya_set_cr_lft : Real;
      kyd_cr_ccw : Bool;
      kyd_cr_cw : Bool;
      cw_req : Bool;
      ccw_req : Bool;
   END_VAR
BEGIN


       "BM_SEED_TMP_CTL_DB"();

       //----------------------------------------------------------------------
       //  xtal lift drive
       //----------------------------------------------------------------------
       "PDO".XT_LFT_ENB := TRUE;



       #xt_lft_down_enb := ("LT".V7_OPEN  OR     // xt-lift down enable
                           ("LT".V7_CLOSE  AND "DV".APS_GCH_DELAYED AND ("AV".ACT_XT_POS < "CNF".XT_LO_POS)));

       #kyd_xt_lft_up     := (("KYD".XT_LFT_UP AND NOT "DV".EMG_DRV_ENB) OR     // signal from pc during normal operation     
                            ("KYD".XT_EMG_RAI AND "DV".EMG_DRV_ENB));           // signal from button on op panel in emergency mode

       #kyd_xt_lft_dn     := ("KYD".XT_LFT_DN AND NOT "DV".EMG_DRV_ENB)        // signal from pc during normal operation     
                             AND #xt_lft_down_enb;

       #kyd_xt_lft_fast   := ("KYD".XT_LFT_FST OR 
                            ("DV".EMG_DRV_ENB AND "KYD".XT_EMG_RAI))           // set fast mode in emergency mode
                            AND ((#xt_lft_up AND "DV".XT_LFT_FAST_UP_ENB OR (#xt_lft_dn AND "DV".XT_LFT_FAST_DN_ENB)));                 

       #kyd_xt_lft_stop   := ("KYD".XT_LFT_OFF AND NOT "DV".EMG_DRV_ENB)                           // stop signal from PC only for normal opreration button 
                            OR NOT "PDI".EMO
                            OR "DV".EMG_DVC_OFF                                                 // stop all drives when switching to emergency mode
                            OR ("DV".EMG_DRV_ENB AND NOT "KYD".XT_EMG_RAI)    
                            OR  "DV".EMG_STOP                                                   // stop drive when switching from emergency mode to normal op.
                            OR #xt_lft_dn AND NOT #xt_lft_down_enb;                          // stop lift down when enable flag disapears                                                                


       // xtal downwards
          "CM_ITL_IO"(ADR := 20,
                 KYD_ON := #kyd_xt_lft_dn,
                 KYD_OFF:= #kyd_xt_lft_stop,
                 AUTO := "APC".AUTOMATIC,
                 DC_ON:= "DC".XT_LFT_DN,
                 CON1 := "PDI".EMO AND "DV".MAIN_SWITCH_ON,
                 CON2 := NOT "FLT".DRV_XT_LFT_RUN_FLT,
                 CON3 := NOT "LT".XT_LFT_UP,                         
                 CON4 := "DV".XT_LS_LFT_DN,    
                 CON5 := ("DV".SERVICE OR "LT".XT_LFT_REF_DONE),                       
                 CON6 := NOT "DV".EMG_STOP,
                 CON7 := #xt_lft_down_enb,               
                 CON8 := "SysLog1",
                 ITL_OUT:= "STA_ITL_CAUSE",
                 LT_OUT := #xt_lft_dn);


       // xtal upwards
          "CM_ITL_IO"(ADR := 21,
                 KYD_ON := #kyd_xt_lft_up OR "DV".MAN_XT_LFT_UP,
                 KYD_OFF:= #kyd_xt_lft_stop,
                 AUTO := "APC".AUTOMATIC,
                 DC_ON:= "DC".XT_LFT_UP,
                 CON1 := "PDI".EMO AND "DV".MAIN_SWITCH_ON,
                 CON2 := NOT "FLT".DRV_XT_LFT_RUN_FLT,
                 CON3 := NOT "LT".XT_LFT_DN,                         
                 CON4 := "DV".XT_LS_LFT_UP,    
                 CON5 := ("DV".SERVICE OR "LT".XT_LFT_REF_DONE),                             
                 CON6 := NOT "DV".EMG_STOP, 
                 CON7 := "DIS".ACT_XT_POS > 10.0,
                 CON8 := "SysLog1",
                 ITL_OUT:= "STA_ITL_CAUSE",
                 LT_OUT := #xt_lft_up);


           "LT".XT_LFT_DN := ("LT".XT_LFT_DN AND (#set_spd_xt_lft<>0.0)) OR #xt_lft_dn;  //  LT.XT_LFT_DN := (LT.XT_LFT_DN AND NOT BM_DRV_XT_LFT.Standstill) OR xt_lft_dn;
           "LT".XT_LFT_UP := ("LT".XT_LFT_UP AND (#set_spd_xt_lft<>0.0)) OR #xt_lft_up;  // LT.XT_LFT_UP  := (LT.XT_LFT_UP AND NOT BM_DRV_XT_LFT.Standstill) OR xt_lft_up; 
           "LT".XT_LFT_OFF := NOT #xt_lft_dn AND NOT #xt_lft_up;
           "LT".XT_LFT_FST := ("LT".XT_LFT_UP OR "LT".XT_LFT_DN) AND NOT "APC".AUTOMATIC AND #kyd_xt_lft_fast;

       // Release reference run
       "LT".XT_LFT_REF_RUN  := ("LT".XT_LFT_REF_RUN OR ("KYD".XT_LFT_REF_RUN AND NOT "LT".XT_LFT_REF_DONE)) AND
                              NOT "KYD".XT_LFT_REF_RESET AND NOT #BM_DRV_XT_LFT.Error AND
                              NOT "APC".AUTOMATIC AND ("APC".STATUS=0) AND
                              "PDI".EMO AND "DV".MAIN_SWITCH_ON AND
                              NOT "FLT".DRV_XT_LFT_RUN_FLT AND NOT "DV".EMG_STOP;

       "LT".XT_LFT_REF_DONE := ("LT".XT_LFT_REF_DONE OR #BM_DRV_XT_LFT.Ref_Done) AND 
                             (NOT "KYD".XT_LFT_REF_RESET OR "APC".AUTOMATIC OR ("APC".STATUS<>0)); // AND
                             //((AV.ACT_XT_POS>0.0 AND AV.ACT_XT_POS<4800.0) OR LT.XT_LFT_REF_RUN);                     

       // set crystal lift
       //-----------------
       IF "LT".XT_LFT_FST AND NOT (ABS("CTL".SET_XT_SPD) > "CNF_XT_LFT_LZ950".MAX_SPEED) THEN
           #set_spd_xt_lft_real := ABS("CTL".SET_XT_SPD) * "CNF_XT_LFT_LZ950".RATIO_FST_NRM;    
       ELSE
           #set_spd_xt_lft_real := ABS("CTL".SET_XT_SPD + "CTL".SET_SPEED_OFFS + "AV".MLT_LVL_SFT_OFFS_SPD);    
       END_IF;

       // Track manual set point in automatic mode
       //----------------------------------------
       IF "APC".AUTOMATIC AND NOT "LT".SMI_XT_SPD_ON OR ("CTL".SET_SPEED_OFFS <> 0.0) THEN   //track KYA variable always when output of offset speed controller for gap control is unequal zero                             
           "KYA".SET_XT_SPD := #set_spd_xt_lft_real;
       END_IF;

       IF "LT".XT_LFT_OFF  THEN
           "KYA".SET_XT_SPD  := 0.0;
       END_IF;

           // Sollwerte rampen
           //-------------------------
           IF "SysTick100ms" THEN
               IF ("DV".XT_LS_LFT_UP OR #xt_lft_dn) AND ("DV".XT_LS_LFT_DN OR #xt_lft_up) AND "PDI".EMO THEN
                   IF ((#set_spd_xt_lft_real-#set_spd_xt_lft) > 12.5)  THEN
                       #set_spd_xt_lft := #set_spd_xt_lft+ 12.5;   // 1000mm/8s =12,5mm/0.1s
                   ELSE
                       IF ((#set_spd_xt_lft_real-#set_spd_xt_lft) < -12.5)  THEN
                           #set_spd_xt_lft := #set_spd_xt_lft - 12.5;   // 1000mm/8s =12,5mm/0.1s
                       ELSE
                           #set_spd_xt_lft := #set_spd_xt_lft_real;
                       END_IF;
                   END_IF;
               ELSE
                   #set_spd_xt_lft := #set_spd_xt_lft_real;
               END_IF;    
           END_IF;

           // Sollwert f黵 Regler aufbereiten
           IF "LT".XT_LFT_UP THEN
               #set_speed_lft := -#set_spd_xt_lft;
           ELSE
              IF "LT".XT_LFT_DN THEN
                  #set_speed_lft := #set_spd_xt_lft;
              ELSE
                  #set_speed_lft := 0.0;
              END_IF;
           END_IF;

       IF "LT".XT_LFT_FST  THEN
          "DIS".SET_XT_SPD := "KYA".SET_XT_SPD * "CNF_XT_LFT_LZ950".RATIO_FST_NRM;
       ELSE
          IF "KYA".SET_XT_SPD> "CNF".XT_LFT_RANGE THEN
             "KYA".SET_XT_SPD := "CNF".XT_LFT_RANGE;
          END_IF;
          "DIS".SET_XT_SPD  := "KYA".SET_XT_SPD;
       END_IF;

       //write display value of effective pull speed
       //-------------------------------------------
       "DIS".SET_EFF_XT_SPD  :=  "KYA".SET_XT_SPD - "CTL".SET_SPEED_OFFS - "AV".MLT_LVL_SFT_OFFS_SPD;  //variable used in logging

       // Motor controller control                                                                        
       #BM_DRV_XT_LFT(Enable      := INT_TO_BOOL("CNF_XT_LFT_LZ950".CTRL_ACTIV) AND ("LT".XT_LFT_UP OR "LT".XT_LFT_DN OR "LT".XT_LFT_REF_RUN), 
                   Pro_start     := "LT".XT_LFT_UP OR "LT".XT_LFT_DN,   
                   Speed_ext_ovr := TRUE,   
                   Ref_Start     := "LT".XT_LFT_REF_RUN, 
                   Ref_reset     := "KYD".XT_LFT_REF_RESET AND NOT "APC".AUTOMATIC AND ("APC".STATUS=0),
                   Reset_error   := "KYD".XT_LFT_TRIP_RES,
                   Stop          := NOT "LT".XT_LFT_UP AND NOT "LT".XT_LFT_DN,
                   Profil        := "CNF_XT_LFT_LZ950".Profil,
                   PM_ADR_E      := INT_TO_WORD("CNF_XT_LFT_LZ950".PE_ADR),                                    
                   PM_ADR_A      := INT_TO_WORD("CNF_XT_LFT_LZ950".PA_ADR),                
                   Units_per_rev := "CNF_XT_LFT_LZ950".UNITS_PER_REV,                       
                   Gear_ratio    := "CNF_XT_LFT_LZ950".FEED_CONST,
                   Set_vel       := #set_speed_lft); 


       //actual motor values
       //---------------------
       "AV".ACT_XT_POS   := #BM_DRV_XT_LFT.Act_pos;   
       "DIS".ACT_XT_POS  := "AV".ACT_XT_POS;   

       IF "LT".XT_LFT_UP XOR "LT".XT_LFT_DN THEN
               "DIS".ACT_XT_SPD  := ABS(#BM_DRV_XT_LFT.Act_vel);
          ELSE
               "DIS".ACT_XT_SPD  := 0.0;
       END_IF;

       IF "PAR_MAIN".MCONST_LIM_XTAL_UP < "CNF".xt_high_pos THEN
          "PAR_MAIN".MCONST_LIM_XTAL_UP := "CNF".xt_high_pos;
       END_IF;   
       "DV".XT_LS_LFT_UP := ("AV".ACT_XT_POS > "PAR_MAIN".MCONST_LIM_XTAL_UP) OR ("PDI".KEY_XT_LFT_SRV AND NOT "PDI".LS_XT_SFT_SRV_POS AND ("APC".STATUS=0));
         IF "PAR_MAIN".MCONST_LIM_XTAL_DN> "CNF".xt_low_pos THEN
          "PAR_MAIN".MCONST_LIM_XTAL_DN := "CNF".xt_low_pos;
       END_IF;   
       "DV".XT_LS_LFT_DN := "AV".ACT_XT_POS < "PAR_MAIN".MCONST_LIM_XTAL_DN;
       "DV".XT_LFT_FAST_UP_ENB := ("AV".ACT_XT_POS > ("PAR_MAIN".MCONST_LIM_XTAL_UP + "CNF".xt_lft_rmp));
       "DV".XT_LFT_FAST_DN_ENB := ("LT".V7_OPEN AND "AV".ACT_XT_POS < ("PAR_MAIN".MCONST_LIM_XTAL_DN - "CNF".xt_lft_rmp))  OR  ("PDI".LS_V7_SW_IN AND ("AV".ACT_XT_POS < ("CNF".XT_LO_POS - "CNF".xt_lft_rmp)));


        //actual fault
       //---------------------
       "DIS".XT_LFT_ERR_CODE     := #BM_DRV_XT_LFT.Error_code;     // Fehlernummer Umrichter
       "FLT".DRV_XT_LFT_RUN_FLT  := #BM_DRV_XT_LFT.Error;                // Fehlerbit Umrichter
       "FLT".DRV_XT_LFT_PAR_FLT  := FALSE;
       "FLT".XT_LFT_POS_REF      := NOT "LT".XT_LFT_REF_DONE;                       // Antrieb nicht referenziert
       "FLT".XT_LFT_SW_LIMIT     := NOT ("DV".XT_LS_LFT_UP AND "DV".XT_LS_LFT_DN) AND // Fehler Antrieb nicht in Grenzparametern
                                  NOT "LT".XT_LFT_REF_RUN;
       "FLT".XT_SLS              := #BM_DRV_XT_LFT.LS_neg OR #BM_DRV_XT_LFT.LS_pos;  // Fehler Sicherheitsendschalter
       //FLT.XT_TOP_POS          :=  NOT PDI.XT_TOP_POS AND NOT LT.XT_LFT_REF_RUN;      // seed holder switch

       IF "LT".V7_CLOSE  AND NOT "LT".V7_OPEN AND ("AV".ACT_XT_POS >= "CNF".XT_LO_POS) THEN
           IF (("KYD".XT_LFT_DN OR "DC".XT_LFT_DN) OR "PDO".XT_LFT_ENB) THEN
               "FLT".V7_CLOSED  := TRUE;
           END_IF;
       ELSE
           "FLT".V7_CLOSED  := FALSE;
       END_IF;        

       IF "DV".EMG_DRV_ENB THEN
          IF "KYD".XT_EMG_RAI THEN
             "KYA".SET_XT_SPD := "CNF".XT_LFT_SPEED_FAST/"CNF_XT_LFT_LZ950".RATIO_FST_NRM; // setpoint XT_lift:= 50 mm/min in emergency mode (fast mode active)
          ELSE
             "KYA".SET_XT_SPD := 0.0;
          END_IF;
       END_IF;

       //------- xtal rotation ------------------------------------------------------------
       // xtal rotation
          "PDO".XT_ROT_ENB := TRUE; 

          "CM_ITL_IO"(ADR := 22,
                 KYD_ON := "KYD".XT_ROT_CW AND NOT "DV".EMG_DRV_ENB,
                 KYD_OFF:= "KYD".XT_ROT_OFF OR "DV".PWR_FAIL_XT_ROT_OFF OR "DV".EMG_DVC_OFF,
                 AUTO := "APC".AUTOMATIC AND NOT "SY".CTL_XT_ROT_SMI,
                 DC_ON:= "DC".XT_ROT_CW,
                 CON1 := "PDI".EMO,
                 CON2 := NOT "FLT".DRV_XT_ROT_RUN_FLT,
                 CON3 := NOT "LT".XT_ROT_CCW,                         
                 CON4 := NOT "DV".PWR_FAIL_XT_ROT_OFF,    
                 CON5 := NOT "DV".EMG_DVC_OFF,               
                 CON6 := "SysLog1",
                 CON7 := "SysLog1",                       
                 CON8 := "SysLog1",
                 ITL_OUT:= "STA_ITL_CAUSE",
                 LT_OUT := #xt_rot_cw);

         "CM_ITL_IO"(ADR := 23,
                 KYD_ON := "KYD".XT_ROT_CCW AND NOT "DV".EMG_DRV_ENB,
                 KYD_OFF:= "KYD".XT_ROT_OFF OR "DV".PWR_FAIL_XT_ROT_OFF OR "DV".EMG_DVC_OFF,
                 AUTO := "APC".AUTOMATIC AND NOT "SY".CTL_XT_ROT_SMI,
                 DC_ON:= "DC".XT_ROT_CCW,
                 CON1 := "PDI".EMO,
                 CON2 := NOT "FLT".DRV_XT_ROT_RUN_FLT,
                 CON3 := NOT "LT".XT_ROT_CW,                         
                 CON4 := NOT "DV".PWR_FAIL_XT_ROT_OFF,    
                 CON5 := NOT "DV".EMG_DVC_OFF,               
                 CON6 := "SysLog1",
                 CON7 := "SysLog1",                       
                 CON8 := "SysLog1",
                 ITL_OUT:= "STA_ITL_CAUSE",
                 LT_OUT := #xt_rot_ccw);


           "LT".XT_ROT_CW  := ("LT".XT_ROT_CW AND NOT #BM_DRV_XT_ROT.Standstill) OR #xt_rot_cw;       
           "LT".XT_ROT_CCW := ("LT".XT_ROT_CCW AND NOT #BM_DRV_XT_ROT.Standstill) OR #xt_rot_ccw;
           "LT".XT_ROT_OFF := NOT #xt_rot_cw AND NOT #xt_rot_ccw;

       // setpoints
       //--------------------
       #set_spd_xt_rot_real := "CM_INSELECT" ( auto   := ("APC".AUTOMATIC AND NOT "SY".CTL_XT_ROT_SMI),        
                                            track  := TRUE,
                                            ac     := "AC".SET_XT_ROT,                
                                            kya    := "KYA".SET_XT_ROT);
       IF "KYA".SET_XT_ROT> "CNF".XT_ROT_RANGE THEN
          "KYA".SET_XT_ROT := "CNF".XT_ROT_RANGE;
       END_IF;
       IF "LT".XT_ROT_OFF  THEN
           "KYA".SET_XT_ROT  := 0.0;
       END_IF;


       // Sollwerte rampen
       //-------------------------
       IF "SysTick1s" THEN
           IF ((#set_spd_xt_rot_real-#set_spd_xt_rot) > 0.3)  THEN
               #set_spd_xt_rot := #set_spd_xt_rot+ 0.02917;   // 35rpm/1200s = 0.29167
           ELSE
               IF ((#set_spd_xt_rot_real-#set_spd_xt_rot) < -0.3)  THEN
                   #set_spd_xt_rot := #set_spd_xt_rot - 0.02917;   // 35rpm/1200s = 0.29167
               ELSE
                   #set_spd_xt_rot := #set_spd_xt_rot_real;
               END_IF;
           END_IF;
       END_IF;

           // Sollwert f黵 Regler aufbereiten
       IF "LT".XT_ROT_CW THEN
           #set_speed_rot := #set_spd_xt_rot;
       ELSE
           IF "LT".XT_ROT_CCW THEN
               #set_speed_rot := -#set_spd_xt_rot;
           ELSE
               #set_speed_rot := 0.0;
           END_IF;
       END_IF;


       // Motor controller control                                                                        
       #BM_DRV_XT_ROT(Enable      :=("LT".XT_ROT_CW OR "LT".XT_ROT_CCW), 
                   Pro_start     := #BM_DRV_XT_ROT.Ref_Done AND("LT".XT_ROT_CW OR "LT".XT_ROT_CCW) ,   
                   Speed_ext_ovr := TRUE,   
                   Ref_Start     := #BM_DRV_XT_ROT.Ready AND NOT #BM_DRV_XT_ROT.Ref_Done, 
                   Ref_reset     := FALSE,
                   Reset_error   := "KYD".XT_ROT_TRIP_RES,
                   Stop          := NOT "LT".XT_ROT_CW AND NOT "LT".XT_ROT_CCW,
                   Profil        := "CNF_XT_ROT_LZ950".Profil,
                   PM_ADR_E      := INT_TO_WORD("CNF_XT_ROT_LZ950".PE_ADR),                                    
                   PM_ADR_A      := INT_TO_WORD("CNF_XT_ROT_LZ950".PA_ADR),                
                   Units_per_rev := "CNF_XT_ROT_LZ950".UNITS_PER_REV,                       
                   Gear_ratio    := "CNF_XT_ROT_LZ950".GEAR_RATIO_Z/"CNF_XT_ROT_LZ950".GEAR_RATIO_N,
                   Set_vel       := #set_speed_rot); 

        //   KYD.XT_ROT_TRIP_RES := DC.RES_ERR_DRV_XT_ROT;

       //actual motor values
       //---------------------
       IF "LT".XT_ROT_CW XOR "LT".XT_ROT_CCW THEN
               "DIS".ACT_XT_ROT  := ABS(#BM_DRV_XT_ROT.Act_vel);
          ELSE
               "DIS".ACT_XT_ROT  := 0.0;
       END_IF;

       "DIS".SET_XT_ROT  := "KYA".SET_XT_ROT;

       //actual fault
       //---------------------
       "DIS".XT_ROT_ERR_CODE     := #BM_DRV_XT_ROT.Error_code;     // Fehlernummer Umrichter
       "FLT".DRV_XT_ROT_RUN_FLT  := #BM_DRV_XT_ROT.Error;                // Fehlerbit Umrichter
       "FLT".DRV_XT_ROT_PAR_FLT  := FALSE;


       //----------------------------------------------------------------------------------
       //crucible lift
       //----------------------------------------------------------------------------------
       "PDO".CR_LFT_ENB :=  TRUE;     //(cr_lft_up XOR cr_lft_dn) OR LT.CR_LFT_REF_RUN OR LT.CR_LFT_REL_LS OR NOT BM_DRV_CR_LFT.Standstill;


       #kyd_cr_lft_up     := ("KYD".CR_LFT_UP AND NOT "DV".EMG_DRV_ENB);        // signal from pc during normal operation     

       #kyd_cr_lft_dn     := (("KYD".CR_LFT_DN AND NOT "DV".EMG_DRV_ENB) OR     // signal from pc during normal operation     
                            ("KYD".CR_EMG_LOW AND "DV".EMG_DRV_ENB));           // signal from button on op panel in emergency mode 
                            //AND cr_lft_down_enb;  !!!!

       #kyd_cr_lft_fast   := ("KYD".CR_LFT_FST OR 
                            ("DV".EMG_DRV_ENB AND "KYD".CR_EMG_LOW))          // set fast mode in emergency mode
                            AND ((#cr_lft_up AND "DV".CR_LFT_FAST_UP_ENB 
                            OR (#cr_lft_dn AND "DV".CR_LFT_FAST_DN_ENB)));                 

       #kyd_cr_lft_stop   := ("KYD".CR_LFT_OFF AND NOT "DV".EMG_DRV_ENB)                           // stop signal from PC only for normal opreration button 
                            OR NOT "PDI".EMO
                            OR "DV".EMG_DVC_OFF                                                 // stop all drives when switching to emergency mode
                            OR ("DV".EMG_DRV_ENB AND NOT "KYD".CR_EMG_LOW)    
                            OR  "DV".EMG_STOP;                                                  // stop drive when switching from emergency mode to normal op.
                          //  OR cr_lft_dn AND NOT cr_lft_down_enb;                          // stop lift down when enable flag disapears                                                                


       // crucible downwards
          "CM_ITL_IO"(ADR := 24,
                 KYD_ON := #kyd_cr_lft_dn,
                 KYD_OFF:= #kyd_cr_lft_stop,
                 AUTO := "APC".AUTOMATIC,
                 DC_ON:= "DC".CR_LFT_DN,
                 CON1 := "PDI".EMO AND "DV".MAIN_SWITCH_ON,
                 CON2 := NOT "FLT".DRV_CR_LFT_RUN_FLT,
                 CON3 := NOT "LT".CR_LFT_UP,                         
                 CON4 := "DV".CR_LS_LFT_DN,  
                 CON5 := ("DV".SERVICE OR "LT".CR_LFT_REF_DONE),                       
                 CON6 := NOT "DV".EMG_STOP,
                 CON7 := "SysLog1",               
                 CON8 := "SysLog1",
                 ITL_OUT:= "STA_ITL_CAUSE",
                 LT_OUT := #cr_lft_dn);


       // crucible upwards
          "CM_ITL_IO"(ADR := 25,
                 KYD_ON := #kyd_cr_lft_up OR "DV".MAN_CR_LFT_UP,
                 KYD_OFF:= #kyd_cr_lft_stop,
                 AUTO := "APC".AUTOMATIC,
                 DC_ON:= "DC".CR_LFT_UP,
                 CON1 := "PDI".EMO AND "DV".MAIN_SWITCH_ON,
                 CON2 := NOT "FLT".DRV_CR_LFT_RUN_FLT,
                 CON3 := NOT "LT".CR_LFT_DN,                         
                 CON4 := "DV".CR_LS_LFT_UP,    
                 CON5 := ("DV".SERVICE OR "LT".CR_LFT_REF_DONE),                       
                 CON6 := NOT "DV".EMG_STOP,
                 CON7 := "SysLog1",
                 CON8 := "SysLog1",
                 ITL_OUT:= "STA_ITL_CAUSE",
                 LT_OUT := #cr_lft_up);

           //LT.CR_LFT_UP := (LT.CR_LFT_UP AND NOT BM_DRV_CR_LFT.Standstill) OR cr_lft_up;                         
           //LT.CR_LFT_DN := (LT.CR_LFT_DN AND NOT BM_DRV_CR_LFT.Standstill) OR cr_lft_dn; 
           "LT".CR_LFT_UP := ("LT".CR_LFT_UP AND (#set_spd_cr_lft <> 0.0)) OR #cr_lft_up;                         
           "LT".CR_LFT_DN := ("LT".CR_LFT_DN AND (#set_spd_cr_lft <> 0.0)) OR #cr_lft_dn; 
           "LT".CR_LFT_OFF := NOT #cr_lft_dn AND NOT #cr_lft_up;

           "LT".CR_LFT_FST := ((NOT "APC".AUTOMATIC AND #kyd_cr_lft_fast) OR
                            ("APC".AUTOMATIC AND (ABS("CTL".SET_CR_SPD)> "CNF_CR_LFT_LZ950".MAX_SPEED)
                            AND ((#cr_lft_up AND "DV".CR_LFT_FAST_UP_ENB) OR (#cr_lft_dn AND "DV".CR_LFT_FAST_DN_ENB))))
                            AND (#cr_lft_up OR #cr_lft_dn);

        // Release reference run
        "LT".CR_LFT_REF_RUN := (("LT".CR_LFT_REF_RUN OR "KYD".CR_LFT_REF_RUN) AND NOT "LT".CR_LFT_REF_DONE) AND
                              NOT "KYD".CR_LFT_REF_RESET AND NOT #BM_DRV_CR_LFT.Error AND
                              NOT "APC".AUTOMATIC AND ("APC".STATUS=0) AND
                              "PDI".EMO AND "DV".MAIN_SWITCH_ON AND 
                              NOT "FLT".DRV_CR_LFT_RUN_FLT AND NOT "DV".EMG_STOP;

        "LT".CR_LFT_REF_DONE    := ("LT".CR_LFT_REF_DONE OR #BM_DRV_CR_LFT.Ref_Done) AND 
                                 (NOT "KYD".CR_LFT_REF_RESET OR "APC".AUTOMATIC OR ("APC".STATUS<>0)); // AND    
                                 //((AV.ACT_CR_POS>0.0 AND AV.ACT_CR_POS<1060.0) OR LT.CR_LFT_REF_RUN);                     

       // set point crucible lift
       //------------------------   
       IF "KYA".SET_CR_SPD >"CNF_CR_LFT_LZ950".MAX_SPEED THEN
           "KYA".SET_CR_SPD := "CNF_CR_LFT_LZ950".MAX_SPEED;
       END_IF;     

       IF "LT".CR_LFT_FST AND NOT(ABS("CTL".SET_CR_SPD)> "CNF_CR_LFT_LZ950".MAX_SPEED) THEN
           #set_spd_cr_lft_real := ABS("CTL".SET_CR_SPD) * "CNF_CR_LFT_LZ950".RATIO_FST_NRM;
       ELSE
           IF "LT".CR_LFT_OFF THEN
              #set_spd_cr_lft_real := 0.0;
           ELSE
              #set_spd_cr_lft_real := ABS("CTL".SET_CR_SPD + "CTL".SET_SPEED_OFFS + "AV".MLT_LVL_SFT_OFFS_SPD);
           END_IF;
       END_IF;

       // Track manual set point in automatic mode
       //----------------------------------------
       IF "APC".AUTOMATIC AND NOT "LT".SMI_CR_SPD_ON OR ("CTL".SET_SPEED_OFFS <> 0.0) THEN   //track KYA variable always when output of offset speed controller for gap control is unequal zero 
           "KYA".SET_CR_SPD := #set_spd_cr_lft_real;
       END_IF;

       IF "LT".CR_LFT_OFF  THEN
          "KYA".SET_CR_SPD  := 0.0;
       END_IF;

        IF "SysTick100ms" THEN
           IF ("DV".CR_LS_LFT_DN OR #cr_lft_up) AND ("DV".CR_LS_LFT_UP OR #cr_lft_dn) AND "PDI".EMO THEN
               IF ((#set_spd_cr_lft_real-#set_spd_cr_lft) > 5.0) THEN
                   #set_spd_cr_lft := #set_spd_cr_lft+5.0;         //   200mm/min 4s => 5mm/0.1s
               ELSE
                   IF ((#set_spd_cr_lft_real-#set_spd_cr_lft) < -5.0) THEN
                       #set_spd_cr_lft := #set_spd_cr_lft-5.0;
                   ELSE
                       #set_spd_cr_lft := #set_spd_cr_lft_real;
                   END_IF;
               END_IF;
           ELSE
               #set_spd_cr_lft := #set_spd_cr_lft_real;
           END_IF;
        END_IF;

        IF "LT".CR_LFT_UP THEN
           #set_speed_cr_lft := #set_spd_cr_lft;
        ELSE
           IF "LT".CR_LFT_DN THEN
              #set_speed_cr_lft := -#set_spd_cr_lft;
           ELSE
              #set_speed_cr_lft := 0.0;
           END_IF;
        END_IF;

       //write display value of crucible speed set point
       //-----------------------------------------------
       IF "LT".CR_LFT_FST  THEN
           "DIS".SET_CR_SPD := "KYA".SET_CR_SPD * "CNF_CR_LFT_LZ950".RATIO_FST_NRM;
       ELSE
           IF ("KYA".SET_CR_SPD > "CNF".CR_LFT_RANGE) THEN
               "KYA".SET_CR_SPD := "CNF".CR_LFT_RANGE;
           END_IF;
           "DIS".SET_CR_SPD  := "KYA".SET_CR_SPD;
       END_IF;

        // Motor controller control                                                                        
        #BM_DRV_CR_LFT(Enable      := INT_TO_BOOL("CNF_CR_LFT_LZ950".CTRL_ACTIV) AND ("LT".CR_LFT_UP OR "LT".CR_LFT_DN OR "LT".CR_LFT_REF_RUN), 
                    Pro_start     := "LT".CR_LFT_UP OR "LT".CR_LFT_DN,   
                    Speed_ext_ovr := TRUE,   
                    Ref_Start     := "LT".CR_LFT_REF_RUN, 
                    Ref_reset     := "KYD".CR_LFT_REF_RESET AND NOT "APC".AUTOMATIC AND ("APC".STATUS=0),
                    Reset_error   := "KYD".CR_LFT_TRIP_RES,
                    Stop          := NOT "LT".CR_LFT_UP AND NOT "LT".CR_LFT_DN,
                    Profil        := "CNF_CR_LFT_LZ950".Profil,
                    PM_ADR_E      := INT_TO_WORD("CNF_CR_LFT_LZ950".PE_ADR),                                    
                    PM_ADR_A      := INT_TO_WORD("CNF_CR_LFT_LZ950".PA_ADR),                
                    Units_per_rev := "CNF_CR_LFT_LZ950".UNITS_PER_REV,                       
                    Gear_ratio    := "CNF_CR_LFT_LZ950".FEED_CONST,
                    Set_vel       := #set_speed_cr_lft); 


        //actual motor values
        //---------------------
        "AV".ACT_CR_POS   := #BM_DRV_CR_LFT.Act_pos;   
        "DIS".ACT_CR_POS  := "AV".ACT_CR_POS;   

        IF "LT".CR_LFT_UP XOR "LT".CR_LFT_DN THEN
               "DIS".ACT_CR_SPD  := ABS(#BM_DRV_CR_LFT.Act_vel);
           ELSE
               "DIS".ACT_CR_SPD  := 0.0;
        END_IF;

        IF "PAR_MAIN".MCONST_LIM_CR_UP> "CNF".cr_high_pos THEN
           "PAR_MAIN".MCONST_LIM_CR_UP := "CNF".cr_high_pos;
        END_IF;   
        "DV".CR_LS_LFT_UP := "AV".ACT_CR_POS < "PAR_MAIN".MCONST_LIM_CR_UP;
        IF "PAR_MAIN".MCONST_LIM_CR_DN< "CNF".cr_low_pos THEN
           "PAR_MAIN".MCONST_LIM_CR_DN := "CNF".cr_low_pos;
        END_IF;       
        "DV".CR_LS_LFT_DN := "AV".ACT_CR_POS > "PAR_MAIN".MCONST_LIM_CR_DN;
        "DV".CR_LFT_FAST_UP_ENB := ("AV".ACT_CR_POS < ("PAR_MAIN".MCONST_LIM_CR_UP - "CNF".cr_lft_rmp));
        "DV".CR_LFT_FAST_DN_ENB :=  ("AV".ACT_CR_POS > ("PAR_MAIN".MCONST_LIM_CR_DN + "CNF".cr_lft_rmp));



        //actual fault
        //---------------------
        "DIS".CR_LFT_ERR_CODE     := #BM_DRV_CR_LFT.Error_code;     // Fehlernummer Umrichter
        "FLT".DRV_CR_LFT_RUN_FLT  := #BM_DRV_CR_LFT.Error;                // Fehlerbit Umrichter
        "FLT".DRV_CR_LFT_PAR_FLT  := FALSE;
        "FLT".CR_LFT_POS_REF      := NOT "LT".CR_LFT_REF_DONE;                       // Antrieb nicht referenziert
        "FLT".CR_LFT_SW_LIMIT     := NOT ("DV".CR_LS_LFT_UP AND "DV".CR_LS_LFT_DN) AND // Fehler Antrieb nicht in Grenzparametern
                                   NOT "LT".CR_LFT_REF_RUN;
        "FLT".CR_SLS              := #BM_DRV_CR_LFT.LS_neg OR #BM_DRV_CR_LFT.LS_pos;  // Fehler Sicherheitsendschalter


        IF "DV".EMG_DRV_ENB THEN
            IF "KYD".CR_EMG_LOW THEN
                "KYA".SET_CR_SPD := "CNF".CRUC_LFT_SPEED_FAST/"CNF_CR_LFT_LZ950".RATIO_FST_NRM; // setpoint cr_lift:= 50 mm/min in emergency mode (fast mode active)
            ELSE
                "KYA".SET_CR_SPD := 0.0;
            END_IF;
        END_IF;

       //----------------------------------------------------------------------------------
       //crucible rotation
       //----------------------------------------------------------------------------------
       //set enable output
       //-----------------
       "PDO".CR_ROT_ENB :=  TRUE;

          "CM_ITL_IO"(ADR := 26,
                 KYD_ON := "KYD".CR_ROT_CW,
                 KYD_OFF:= "KYD".CR_ROT_OFF,
                 AUTO := "APC".AUTOMATIC AND NOT "SY".CTL_CR_ROT_SMI,
                 DC_ON:= "DC".CR_ROT_CW,
                 CON1 := "PDI".EMO,
                 CON2 := NOT "FLT".DRV_CR_ROT_RUN_FLT,
                 CON3 := NOT "LT".CR_ROT_CCW,                         
                 CON4 := NOT "DV".EMG_DRV_ENB,    
                 CON5 := NOT "DV".EMG_DVC_OFF,               
                 CON6 := "SysLog1",
                 CON7 := "SysLog1",                       
                 CON8 := "SysLog1",
                 ITL_OUT:= "STA_ITL_CAUSE",
                 LT_OUT := #cr_rot_cw);

         "CM_ITL_IO"(ADR := 27,
                 KYD_ON := "KYD".CR_ROT_CCW,
                 KYD_OFF:= "KYD".CR_ROT_OFF,
                 AUTO := "APC".AUTOMATIC AND NOT "SY".CTL_CR_ROT_SMI,
                 DC_ON:= "DC".CR_ROT_CCW,
                 CON1 := "PDI".EMO,
                 CON2 := NOT "FLT".DRV_CR_ROT_RUN_FLT,
                 CON3 := NOT "LT".CR_ROT_CW,                         
                 CON4 := NOT "DV".EMG_DRV_ENB,    
                 CON5 := NOT "DV".EMG_DVC_OFF,               
                 CON6 := "SysLog1",
                 CON7 := "SysLog1",                       
                 CON8 := "SysLog1",
                 ITL_OUT:= "STA_ITL_CAUSE",
                 LT_OUT := #cr_rot_ccw);

           "LT".CR_ROT_CW  := ("LT".CR_ROT_CW AND ("DIS".ACT_CR_ROT<>0.0)) OR #cr_rot_cw;   // NOT BM_DRV_CR_ROT.Standstill    
           "LT".CR_ROT_CCW := ("LT".CR_ROT_CCW AND ("DIS".ACT_CR_ROT<>0.0)) OR #cr_rot_ccw;   //NOT BM_DRV_CR_ROT.Standstill
           "LT".CR_ROT_OFF := NOT #cr_rot_cw AND NOT #cr_rot_ccw;


       // setpoints
       //--------------------
       IF ("APC".STATUS = "APC".SHOULDER) AND ("PAR_MAIN".SH_CRUC_ROT_CTL_ON = 1.0)  OR
          ("APC".STATUS = "APC".BODY) AND ("PAR_MAIN".BY_CRUC_ROT_CTL_ON = 1.0)      THEN
           #ac_in               := "CTL".SET_CR_ROT;  //setpoint comes from control loop
           #cruc_rot_ctl        := TRUE;            //status flag crucible rotation control
       ELSE
           #ac_in               := "AC".SET_CR_ROT;   //setpoint comes from parameter table
           #cruc_rot_ctl        := FALSE;           //status flag crucible rotation control        
       END_IF;        

       //check if crucible rotation oscillation is requested
       //---------------------------------------------------
       IF "APC".AUTOMATIC                            //automatic mode active?
           AND NOT "SY".CTL_CR_ROT_SMI               //semi mode disabled?
           AND NOT #cruc_rot_ctl                    //crucible rotation control disabled?
           AND NOT "DV".CR_ROT_CTL_OFFS_RP           //crucible rotation control flag
           AND ("AC".SET_CR_ROT_OFS > 0.0) THEN      //offset requested?
           #cr_rot_osci_req     := TRUE;            //enable flag for crucible rotation oscillation
       ELSE
           #cr_rot_osci_req     := FALSE;
       END_IF;    

       //calculate time for adding and deducting the offset 
       //--------------------------------------------------


       IF #cr_rot_osci_req THEN                  //rotation offset requested

           IF "SysTick100ms" THEN                 // calculate in 0.1 s steps
               "AV".CR_ROT_OFFS_TIME := "AV".CR_ROT_OFFS_TIME + 0.1;

               IF "DV".CR_ROT_OFFS_ON THEN            
                   #set_cr_rot_ofs := "AC".SET_CR_ROT_OFS;            // for rot value + offset

                   IF ("AV".CR_ROT_OFFS_TIME >= "AC".SET_CR_ROT_ON_TME) THEN
                       "AV".CR_ROT_OFFS_TIME := 0.0;
                       "DV".CR_ROT_OFFS_ON   := FALSE;
                   END_IF;                
               ELSE
                   #set_cr_rot_ofs := - "AC".SET_CR_ROT_OFS;          // for rot value - offset

                   IF ("AV".CR_ROT_OFFS_TIME >= "AC".SET_CR_ROT_OFF_TME) THEN
                       "AV".CR_ROT_OFFS_TIME := 0.0;
                       "DV".CR_ROT_OFFS_ON   := TRUE;
                   END_IF;
               END_IF;        
           END_IF;
       ELSE
           #set_cr_rot_ofs      := 0.0;
           "AV".CR_ROT_OFFS_TIME := 0.0;
           "DV".CR_ROT_OFFS_ON   := FALSE;
       END_IF;    

       //calculate crucible rotation setpoint
       //------------------------------------
       #cr_rot_set := #set_cr_rot_ofs + "CM_INSELECT" (auto   := ("APC".AUTOMATIC AND NOT "SY".CTL_CR_ROT_SMI),        
                                                   track  := FALSE,
                                                   ac     := #ac_in,                
                                                   kya    := "KYA".SET_CR_ROT);

       //check limits of calculated rotation setpoint
       //--------------------------------------------
       IF #cr_rot_set > "CNF".CR_ROT_RANGE THEN
           #cr_rot_set := "CNF".CR_ROT_RANGE;     //set to upper limit
           "KYA".SET_CR_ROT := "CNF".CR_ROT_RANGE;
       END_IF;
       IF #cr_rot_set < 0.0 THEN
           #cr_rot_set := 0.0;                  //set to lower limit
       END_IF;;


       //eliminate crucible rotation setpoint offset if control loop active in shoulder and passive in body
       //--------------------------------------------------------------------------------------------------
       IF ("PAR_MAIN".SH_CRUC_ROT_CTL_ON = 1.0)  AND
          ("APC".STATUS = "APC".BODY)              AND
          ("PAR_MAIN".BY_CRUC_ROT_CTL_ON = 0.0)  AND
          "DV".CR_ROT_CTL_OFFS_RP                    THEN    //cruc rot control flag is set in initialisation of body sequence

           IF "SysTick100ms" THEN                            //call ramp function every 100ms

               "CM_SET_RAMP"(rp_enb      := "DV".CR_ROT_CTL_OFFS_RP,
                           i           := "DV".CR_ROT_OFFS_RP_START,
                           max_dev     := 0.0,
                           rp_start    := 0.0,
                           rp_grad     := "PAR_MAIN".BY_CRUC_ROT_OFFS_RP_GRAD,
                           tme_base    := 60.0,
                           tc_in       := 0.1,
                           set_p       := #cr_rot_set,
                           act_v       := "KYA".SET_CR_ROT,
                           set_out     := "AV".ACT_CR_ROT_SET);
           END_IF;
       ELSE    
           "DV".CR_ROT_CTL_OFFS_RP   := FALSE;               //reset crucible rotation control flag

           //calculate ramp increment in relation to crucible rotation oscillation functionallity 
           //------------------------------------------------------------------------------------
           IF #set_cr_rot_ofs > 0.0 THEN
               IF  "AC".SET_CR_ROT_RP_TME_UP > 0.0 THEN                  //ramp up increment for 100ms with osci fct.    
                   #cr_rot_inc := ("AC".SET_CR_ROT_OFS * 2) / ("AC".SET_CR_ROT_RP_TME_UP * 10);  
               ELSE
                   #cr_rot_inc := "CNF".CR_ROT_RANGE / 1200.0;    //default inc setting if no ramp up time defined
               END_IF;    
           ELSIF #set_cr_rot_ofs < 0.0 THEN
               IF  "AC".SET_CR_ROT_RP_TME_DN > 0.0 THEN                  //ramp down increment for 100ms with osci fct.
                   #cr_rot_inc := ("AC".SET_CR_ROT_OFS * 2) / ("AC".SET_CR_ROT_RP_TME_DN * 10);  
               ELSE
                   #cr_rot_inc := "CNF".CR_ROT_RANGE / 1200.0;    //default inc setting if no ramp down time defined
               END_IF;            
           ELSE    
               #cr_rot_inc := "CNF".CR_ROT_RANGE / 1200.0;    //ramp time 120 sec. from 0 to full rotation range
           END_IF;

           //ramp setpoint for drive controller
           //----------------------------------
           "CM_CYCLE_RAMP"(  ActVal  := "AV".ACT_CR_ROT_SET,           //ramp output value (in/out)
                           SetpVal := #cr_rot_set,                  //setpoint value
                           IncVal  := #cr_rot_inc,                  //increment value
                           TimeFlag:= "SysTick100ms",                //time base 100 ms
                           Enable  := "SysLog1");                   //enable ramp always
       END_IF;            

       //check if oscillation frequency is ok for chosen ramp times
       //----------------------------------------------------------
       IF  #cr_rot_osci_req     THEN 

           IF ("AC".SET_CR_ROT_RP_TME_UP > "AC".SET_CR_ROT_ON_TME)  OR
              ("AC".SET_CR_ROT_RP_TME_DN > "AC".SET_CR_ROT_OFF_TME) OR
              ("AC".SET_CR_ROT_RP_TME_UP = 0.0)                   OR
              ("AC".SET_CR_ROT_RP_TME_DN = 0.0)                   THEN

               "FLT".CR_ROT_OSCI := TRUE;        //set fault message
           ELSE
               "FLT".CR_ROT_OSCI := FALSE;       //reset fault message
           END_IF;    
       ELSE    
           "FLT".CR_ROT_OSCI := FALSE;           //reset fault message
       END_IF;   

       #kya_cruc_rot_set_in     := "AV".ACT_CR_ROT_SET;

       //call device control interface
       //-----------------------------

           IF "LT".CR_ROT_OFF  THEN
               "KYA".SET_CR_ROT    := 0.0;
           ELSIF "APC".AUTOMATIC AND NOT "SY".CTL_CR_ROT_SMI THEN                                
               "KYA".SET_CR_ROT    :=   #kya_cruc_rot_set_in;
           END_IF;

           IF "LT".CR_ROT_CW THEN
               #gear_cr_rot := -1.0; //16384.0 * vk_cr_rot/max_cr_rot_spd;                  
           ELSE
               IF "LT".CR_ROT_CCW THEN
                   #gear_cr_rot := 1.0; //16384.0 * vk_cr_rot/max_cr_rot_spd;                  
               ELSE
                   #gear_cr_rot := 0.0;                  
               END_IF;
           END_IF;

           IF "APC".AUTOMATIC AND NOT "SY".CTL_CR_ROT_SMI THEN
               #set_speed_cr_rot := "AV".ACT_CR_ROT_SET* #gear_cr_rot;
           ELSE
               #set_speed_cr_rot := #kya_cruc_rot_set_in* #gear_cr_rot;
           END_IF;

       // Motor controller control                                                                        
       #BM_DRV_CR_ROT(Enable      := "LT".CR_ROT_CW OR "LT".CR_ROT_CCW, 
                   Pro_start     := #BM_DRV_CR_ROT.Ref_Done AND ("LT".CR_ROT_CW OR "LT".CR_ROT_CCW),   
                   Speed_ext_ovr := TRUE,   
                   Ref_Start     := #BM_DRV_CR_ROT.Ready AND NOT #BM_DRV_CR_ROT.Ref_Done, 
                   Ref_reset     := FALSE,
                   Reset_error   := "KYD".CR_ROT_TRIP_RES,                    
                   Stop          := NOT "LT".CR_ROT_CW AND NOT "LT".CR_ROT_CCW,
                   Profil        := "CNF_CR_ROT_LZ950".Profil,
                   PM_ADR_E      := INT_TO_WORD("CNF_CR_ROT_LZ950".PE_ADR),                                    
                   PM_ADR_A      := INT_TO_WORD("CNF_CR_ROT_LZ950".PA_ADR),                
                   Units_per_rev := "CNF_CR_ROT_LZ950".UNITS_PER_REV,                       
                   Gear_ratio    := "CNF_CR_ROT_LZ950".GEAR_RATIO_Z/"CNF_CR_ROT_LZ950".GEAR_RATIO_N,
                   Set_vel       := #set_speed_cr_rot); 


       //actual motor values
       //---------------------
      IF "LT".CR_ROT_CW XOR "LT".CR_ROT_CCW THEN
               "DIS".ACT_CR_ROT  := ABS(#BM_DRV_CR_ROT.Act_vel);
           ELSE
               "DIS".ACT_CR_ROT  := 0.0;
      END_IF;


       "DIS".SET_CR_ROT  := "AV".ACT_CR_ROT_SET;  //KYA.SET_CR_ROT;

       //actual fault
       //---------------------
       "DIS".CR_ROT_ERR_CODE     := #BM_DRV_CR_ROT.Error_code;     // Fehlernummer Umrichter
       "FLT".DRV_CR_ROT_RUN_FLT  := #BM_DRV_CR_ROT.Error;                // Fehlerbit Umrichter
       "FLT".DRV_CR_ROT_PAR_FLT  := FALSE;
END_FUNCTION_BLOCK

FUNCTION_BLOCK "BM_CALL_HTR_CTRL"   // FB67, SCL
{ S7_Optimized_Access := 'FALSE' }
VERSION : 0.0
// --------------------------------------------------------------------------------
//     program     :    BM_CALL_HTR_CTRL
//     description :    call heater control
//     name        :    G. Eibelsh鋟ser
//     date        :    30.06.2005
// 
//     revision    :    added Injet power supply and TLU earthing monitoring CGS1218
//     name        :    John Wang
//     date        :    15.09.2020
//                     (c)PVATepla AG
//     --------------------------------------------------------------------------------
   VAR
      PM_TLU_HTR_1 : "PM_TLU_PWR_SPL";
      PM_TLU_HTR_2 : "PM_TLU_PWR_SPL";
      PM_INJET_HTR : "PM_INJET_PWR_SPL";
      htr_itl_ok : Bool;
      htr_1_itl_ok : Bool;
      htr_1_on : Bool;
      htr_2_itl_ok : Bool;
      htr_2_on : Bool;
      htr_1_enb : Bool;
      htr_2_enb : Bool;
      start_htr_com : Bool;
      htr_1_pwr_enb_dly : Int;
      htr_2_pwr_enb_dly : Int;
      rst_htr_1_pwr_spl_dly : Int;
      rst_htr_2_pwr_spl_dly : Int;
      com_heater_dly : Int;
      rst_err_htr_eth_dly : Int;
      temp : Array[0..1] of Byte;
      temp_W AT temp : Word;
   END_VAR
   VAR_TEMP
      out_dummy_bool : Bool;
      high_wtr_tmp : Bool;
      high_wtr_tmp_htr_1 : Bool;
      high_wtr_tmp_htr_2 : Bool;
      low_wtr_flw : Bool;
      low_wtr_flw_htr_1 : Bool;
      low_wtr_flw_htr_2 : Bool;
      htr_1_is_on : Bool;
      htr_1_pi_mode : Bool;
      htr_1_pu_mode : Bool;
      htr_1_i_mode : Bool;
      htr_1_u_mode : Bool;
      htr_1_sta_saved : Bool;
      htr_1_flt_i_pri : Bool;
      htr_1_flt_i_max : Bool;
      htr_1_flt_u_max : Bool;
      htr_1_flt_wire : Bool;
      htr_1_flt_flash : Bool;
      htr_1_flt_trafo : Bool;
      htr_1_flt_data_flow : Bool;
      htr_1_flt_data_com : Bool;
      htr_1_flt_data : Bool;
      htr_1_flt_tast : Bool;
      htr_1_flt_ua_max : Bool;
      htr_1_flt_u_min : Bool;
      htr_1_flt_temp : Bool;
      htr_1_flt_sense : Bool;
      htr_1_flt_igbt : Bool;
      htr_1_flt_dioden : Bool;
      htr_1_flt_3 : Bool;
      htr_1_flt_shunt : Bool;
      htr_1_flt_board : Bool;
      htr_1_flt_6 : Bool;
      htr_1_flt_soft : Bool;
      htr_1_flt_timeout : Bool;
      htr_1_flt_short : Bool;
      htr_2_is_on : Bool;
      htr_2_pi_mode : Bool;
      htr_2_pu_mode : Bool;
      htr_2_i_mode : Bool;
      htr_2_u_mode : Bool;
      htr_2_sta_saved : Bool;
      htr_2_flt_i_pri : Bool;
      htr_2_flt_i_max : Bool;
      htr_2_flt_u_max : Bool;
      htr_2_flt_wire : Bool;
      htr_2_flt_flash : Bool;
      htr_2_flt_trafo : Bool;
      htr_2_flt_data_flow : Bool;
      htr_2_flt_data_com : Bool;
      htr_2_flt_data : Bool;
      htr_2_flt_tast : Bool;
      htr_2_flt_ua_max : Bool;
      htr_2_flt_u_min : Bool;
      htr_2_flt_temp : Bool;
      htr_2_flt_sense : Bool;
      htr_2_flt_igbt : Bool;
      htr_2_flt_dioden : Bool;
      htr_2_flt_3 : Bool;
      htr_2_flt_shunt : Bool;
      htr_2_flt_board : Bool;
      htr_2_flt_6 : Bool;
      htr_2_flt_soft : Bool;
      htr_2_flt_timeout : Bool;
      htr_2_flt_short : Bool;
      flt_htr_1_eth_range : Bool;
      flt_htr_1_eth_hw : Bool;
      flt_htr_1_eth_bus : Bool;
      flt_htr_2_eth_range : Bool;
      flt_htr_2_eth_hw : Bool;
      flt_htr_2_eth_bus : Bool;
      flt_pwr_spl_panel_comm : Bool;
      flt_pwr_spl_APF : Bool;
      htr_1_remote : Bool;
      comm_ok : Bool;
      htr_pwr_spl_cool_wtr_flt : Bool;
      htr_pwr_spl_cool_wtr_wrn : Bool;
      htr_1_flt_ctrl : Bool;
      htr_1_flt_comm : Bool;
      htr_1_flt_save : Bool;
      htr_1_flt_ac_pha : Bool;
      htr_1_flt_tmp : Bool;
      htr_1_flt_cur : Bool;
      htr_1_flt_cool_wtr : Bool;
      htr_1_flt_erd_plus : Bool;
      htr_1_flt_erd_min : Bool;
      htr_1_flt_term : Bool;
      htr_1_mod1_flt_syn_kab : Bool;
      htr_1_mod1_flt_sys_tmp : Bool;
      htr_1_mod1_flt_drv : Bool;
      htr_1_mod1_flt_cur : Bool;
      htr_1_mod1_flt_vlt : Bool;
      htr_1_mod1_flt_save : Bool;
      htr_1_mod1_flt_rect : Bool;
      htr_1_mod1_flt_tmp : Bool;
      htr_1_mod2_flt_syn_kab : Bool;
      htr_1_mod2_flt_sys_tmp : Bool;
      htr_1_mod2_flt_drv : Bool;
      htr_1_mod2_flt_cur : Bool;
      htr_1_mod2_flt_vlt : Bool;
      htr_1_mod2_flt_save : Bool;
      htr_1_mod2_flt_rect : Bool;
      htr_1_mod2_flt_tmp : Bool;
      htr_1_mod3_flt_syn_kab : Bool;
      htr_1_mod3_flt_sys_tmp : Bool;
      htr_1_mod3_flt_drv : Bool;
      htr_1_mod3_flt_cur : Bool;
      htr_1_mod3_flt_vlt : Bool;
      htr_1_mod3_flt_save : Bool;
      htr_1_mod3_flt_rect : Bool;
      htr_1_mod3_flt_tmp : Bool;
      htr_1_mod4_flt_syn_kab : Bool;
      htr_1_mod4_flt_sys_tmp : Bool;
      htr_1_mod4_flt_drv : Bool;
      htr_1_mod4_flt_cur : Bool;
      htr_1_mod4_flt_vlt : Bool;
      htr_1_mod4_flt_save : Bool;
      htr_1_mod4_flt_rect : Bool;
      htr_1_mod4_flt_tmp : Bool;
      htr_2_remote : Bool;
      htr_2_flt_ctrl : Bool;
      htr_2_flt_comm : Bool;
      htr_2_flt_save : Bool;
      htr_2_flt_ac_pha : Bool;
      htr_2_flt_tmp : Bool;
      htr_2_flt_cur : Bool;
      htr_2_flt_cool_wtr : Bool;
      htr_2_flt_erd_plus : Bool;
      htr_2_flt_erd_min : Bool;
      htr_2_flt_term : Bool;
      htr_2_mod1_flt_syn_kab : Bool;
      htr_2_mod1_flt_sys_tmp : Bool;
      htr_2_mod1_flt_drv : Bool;
      htr_2_mod1_flt_cur : Bool;
      htr_2_mod1_flt_vlt : Bool;
      htr_2_mod1_flt_save : Bool;
      htr_2_mod1_flt_rect : Bool;
      htr_2_mod1_flt_tmp : Bool;
      htr_2_mod2_flt_syn_kab : Bool;
      htr_2_mod2_flt_sys_tmp : Bool;
      htr_2_mod2_flt_drv : Bool;
      htr_2_mod2_flt_cur : Bool;
      htr_2_mod2_flt_vlt : Bool;
      htr_2_mod2_flt_save : Bool;
      htr_2_mod2_flt_rect : Bool;
      htr_2_mod2_flt_tmp : Bool;
      htr_2_mod3_flt_syn_kab : Bool;
      htr_2_mod3_flt_sys_tmp : Bool;
      htr_2_mod3_flt_drv : Bool;
      htr_2_mod3_flt_cur : Bool;
      htr_2_mod3_flt_vlt : Bool;
      htr_2_mod3_flt_save : Bool;
      htr_2_mod3_flt_rect : Bool;
      htr_2_mod3_flt_tmp : Bool;
      ctrl_high_byte : Byte;
      ctrl_low_byte : Byte;
      low_byte_word_pwr : Word;
      high_byte_word_pwr : Word;
      low_byte_word_cur : Word;
      high_byte_word_cur : Word;
      low_byte_word_sta : Word;
      high_byte_word_sta : Word;
      htr_word_pwr : Word;
      htr_word_cur : Word;
      htr_word_vlt : Word;
      htr_word_sta : Word;
      htr_word_sta_1 : Word;
      ctrl_word : Word;
      set_htr_pwr_dword : DWord;
      set_htr_cur_dword : DWord;
      act_htr_pwr : Real;
      act_htr_cur : Real;
      act_htr_vlt : Real;
      set_htr_pwr : Real;
      set_htr_cur : Real;
      set_htr_vlt : Real;
   END_VAR
BEGIN


